LIN {X 0,Y 312.596,Z 485.644,A -85,B 0,C 180,E1 -15608.66,E2 -15608.66} C_VEL
LIN {X 0,Y 312.546,Z 485.552,A -85,B 0,C 180,E1 -15612.421,E2 -15612.421} C_VEL
LIN {X 0,Y 312.486,Z 485.523,A -85,B 0,C 180,E1 -15616.028,E2 -15616.028} C_VEL
LIN {X 0,Y 312.5,Z 485.561,A -85,B 0,C 180,E1 -15619.874,E2 -15619.874} C_VEL
LIN {X 0,Y 312.531,Z 485.556,A -85,B 0,C 180,E1 -15624.05,E2 -15624.05} C_VEL
LIN {X 0,Y 312.499,Z 485.544,A -85,B 0,C 180,E1 -15627.333,E2 -15627.333} C_VEL
LIN {X 0,Y 312.547,Z 485.546,A -85,B 0,C 180,E1 -15631.275,E2 -15631.275} C_VEL
LIN {X 0,Y 312.58,Z 485.536,A -85,B 0,C 180,E1 -15634.71,E2 -15634.71} C_VEL
LIN {X 0,Y 312.531,Z 485.541,A -85,B 0,C 180,E1 -15638.912,E2 -15638.912} C_VEL
LIN {X 0,Y 312.631,Z 485.51,A -85,B 0,C 180,E1 -15641.656,E2 -15641.656} C_VEL
LIN {X 0,Y 312.687,Z 485.534,A -85,B 0,C 180,E1 -15645.686,E2 -15645.686} C_VEL
LIN {X 0,Y 312.691,Z 485.521,A -85,B 0,C 180,E1 -15649.642,E2 -15649.642} C_VEL
LIN {X 0,Y 312.847,Z 485.516,A -85,B 0,C 180,E1 -15652.254,E2 -15652.254} C_VEL
LIN {X 0,Y 312.712,Z 485.516,A -85,B 0,C 180,E1 -15654.842,E2 -15654.842} C_VEL
LIN {X 0,Y 312.985,Z 485.5,A -85,B 0,C 180,E1 -15658.713,E2 -15658.713} C_VEL
LIN {X 0,Y 313.114,Z 485.481,A -85,B 0,C 180,E1 -15660,E2 -15660} C_VEL
LIN {X 0,Y 312.931,Z 485.487,A -85,B 0,C 180,E1 -15662.575,E2 -15662.575} C_VEL
LIN {X 0,Y 312.886,Z 485.51,A -85,B 0,C 180,E1 -15666.555,E2 -15666.555} C_VEL
LIN {X 0,Y 312.76,Z 485.507,A -85,B 0,C 180,E1 -15669.05,E2 -15669.05} C_VEL
LIN {X 0,Y 312.628,Z 485.542,A -85,B 0,C 180,E1 -15672.991,E2 -15672.991} C_VEL
LIN {X 0,Y 312.632,Z 485.527,A -85,B 0,C 180,E1 -15675.65,E2 -15675.65} C_VEL
LIN {X 0,Y 312.603,Z 485.546,A -85,B 0,C 180,E1 -15679.226,E2 -15679.226} C_VEL
LIN {X 0,Y 312.523,Z 485.543,A -85,B 0,C 180,E1 -15682.782,E2 -15682.782} C_VEL
LIN {X 0,Y 312.597,Z 485.545,A -85,B 0,C 180,E1 -15685.936,E2 -15685.936} C_VEL
LIN {X 0,Y 312.54,Z 485.51,A -85,B 0,C 180,E1 -15689.651,E2 -15689.651} C_VEL
LIN {X 0,Y 312.515,Z 485.544,A -85,B 0,C 180,E1 -15693.69,E2 -15693.69} C_VEL
LIN {X 0,Y 312.516,Z 485.547,A -85,B 0,C 180,E1 -15697.387,E2 -15697.387} C_VEL
LIN {X 0,Y 312.486,Z 485.524,A -85,B 0,C 180,E1 -15700.71,E2 -15700.71} C_VEL
LIN {X 0,Y 312.47,Z 485.562,A -85,B 0,C 180,E1 -15704.207,E2 -15704.207} C_VEL
LIN {X 0,Y 312.483,Z 485.536,A -85,B 0,C 180,E1 -15707.919,E2 -15707.919} C_VEL
LIN {X 0,Y 312.533,Z 485.543,A -85,B 0,C 180,E1 -15711.911,E2 -15711.911} C_VEL
LIN {X 0,Y 312.505,Z 485.487,A -85,B 0,C 180,E1 -15715.791,E2 -15715.791} C_VEL
LIN {X 0,Y 312.524,Z 485.55,A -85,B 0,C 180,E1 -15718.855,E2 -15718.855} C_VEL
LIN {X 0,Y 312.573,Z 485.515,A -85,B 0,C 180,E1 -15721.825,E2 -15721.825} C_VEL
LIN {X 0,Y 312.627,Z 485.658,A -85,B 0,C 180,E1 -15724.403,E2 -15724.403} C_VEL
LIN {X 0,Y 312.857,Z 486.708,A -85,B 0,C 180,E1 -15724.641,E2 -15724.641} C_VEL
LIN {X 0,Y 321.986,Z 506.318,A -85,B 0,C 180,E1 -15725.936,E2 -15725.936} C_VEL
LIN {X 0,Y 324.819,Z 512.869,A -85,B 0,C 180,E1 -15726.326,E2 -15726.326} C_VEL
LIN {X 0,Y 324.111,Z 565.204,A -85,B 0,C 180,E1 -15727.522,E2 -15727.522} C_VEL
LIN {X 0,Y 323.904,Z 578.235,A -85,B 0,C 180,E1 -15728.002,E2 -15728.002} C_VEL
LIN {X 0,Y 323.301,Z 591.093,A -85,B 0,C 180,E1 -15728.731,E2 -15728.731} C_VEL
LIN {X 0,Y 322.411,Z 603.924,A -85,B 0,C 180,E1 -15729.754,E2 -15729.754} C_VEL
LIN {X 0,Y 321.259,Z 614.593,A -85,B 0,C 180,E1 -15730.844,E2 -15730.844} C_VEL
LIN {X 0,Y 319.962,Z 625.427,A -85,B 0,C 180,E1 -15732.256,E2 -15732.256} C_VEL
LIN {X 0,Y 318.575,Z 635.942,A -85,B 0,C 180,E1 -15733.993,E2 -15733.993} C_VEL
LIN {X 0,Y 317.492,Z 643.676,A -85,B 0,C 180,E1 -15735.58,E2 -15735.58} C_VEL
LIN {X 0,Y 316.22,Z 651.351,A -85,B 0,C 180,E1 -15737.518,E2 -15737.518} C_VEL
LIN {X 0,Y 315.27,Z 657.101,A -85,B 0,C 180,E1 -15739.336,E2 -15739.336} C_VEL
LIN {X 0,Y 314.62,Z 661.367,A -85,B 0,C 180,E1 -15741.004,E2 -15741.004} C_VEL
LIN {X 0,Y 313.791,Z 665.259,A -85,B 0,C 180,E1 -15742.924,E2 -15742.924} C_VEL
LIN {X 0,Y 313.2,Z 668.127,A -85,B 0,C 180,E1 -15744.85,E2 -15744.85} C_VEL
LIN {X 0,Y 313.113,Z 669.472,A -85,B 0,C 180,E1 -15746.139,E2 -15746.139} C_VEL
LIN {X 0,Y 312.916,Z 671.03,A -85,B 0,C 180,E1 -15748.713,E2 -15748.713} C_VEL
LIN {X 0,Y 312.881,Z 671.257,A -85,B 0,C 180,E1 -15750,E2 -15750} C_VEL
LIN {X 0,Y 312.979,Z 670.503,A -85,B 0,C 180,E1 -15752.574,E2 -15752.574} C_VEL
LIN {X 0,Y 313.109,Z 669.563,A -85,B 0,C 180,E1 -15753.861,E2 -15753.861} C_VEL
LIN {X 0,Y 313.188,Z 668.259,A -85,B 0,C 180,E1 -15755.15,E2 -15755.15} C_VEL
LIN {X 0,Y 313.784,Z 665.44,A -85,B 0,C 180,E1 -15757.076,E2 -15757.076} C_VEL
LIN {X 0,Y 314.595,Z 661.613,A -85,B 0,C 180,E1 -15758.997,E2 -15758.997} C_VEL
LIN {X 0,Y 315.35,Z 656.533,A -85,B 0,C 180,E1 -15760.984,E2 -15760.984} C_VEL
LIN {X 0,Y 316.401,Z 650.502,A -85,B 0,C 180,E1 -15762.833,E2 -15762.833} C_VEL
LIN {X 0,Y 317.693,Z 642.72,A -85,B 0,C 180,E1 -15764.738,E2 -15764.738} C_VEL
LIN {X 0,Y 319.028,Z 633.047,A -85,B 0,C 180,E1 -15766.641,E2 -15766.641} C_VEL
LIN {X 0,Y 320.237,Z 624.003,A -85,B 0,C 180,E1 -15768.058,E2 -15768.058} C_VEL
LIN {X 0,Y 321.536,Z 613.493,A -85,B 0,C 180,E1 -15769.379,E2 -15769.379} C_VEL
LIN {X 0,Y 322.612,Z 601.973,A -85,B 0,C 180,E1 -15770.533,E2 -15770.533} C_VEL
LIN {X 0,Y 323.532,Z 590.691,A -85,B 0,C 180,E1 -15771.395,E2 -15771.395} C_VEL
LIN {X 0,Y 323.935,Z 578.331,A -85,B 0,C 180,E1 -15772.105,E2 -15772.105} C_VEL
LIN {X 0,Y 324.132,Z 566.47,A -85,B 0,C 180,E1 -15772.554,E2 -15772.554} C_VEL
LIN {X 0,Y 324.608,Z 528.424,A -85,B 0,C 180,E1 -15773.435,E2 -15773.435} C_VEL
LIN {X 0,Y 324.851,Z 512.955,A -85,B 0,C 180,E1 -15773.784,E2 -15773.784} C_VEL
LIN {X 0,Y 316.427,Z 494.129,A -85,B 0,C 180,E1 -15774.953,E2 -15774.953} C_VEL
LIN {X 0,Y 312.807,Z 486.547,A -85,B 0,C 180,E1 -15775.491,E2 -15775.491} C_VEL
LIN {X 0,Y 312.593,Z 485.593,A -85,B 0,C 180,E1 -15775.765,E2 -15775.765} C_VEL
LIN {X 0,Y 312.538,Z 485.545,A -85,B 0,C 180,E1 -15779.65,E2 -15779.65} C_VEL
LIN {X 0,Y 312.519,Z 485.552,A -85,B 0,C 180,E1 -15783.688,E2 -15783.688} C_VEL
LIN {X 0,Y 312.524,Z 485.539,A -85,B 0,C 180,E1 -15787.384,E2 -15787.384} C_VEL
LIN {X 0,Y 312.488,Z 485.554,A -85,B 0,C 180,E1 -15790.708,E2 -15790.708} C_VEL
LIN {X 0,Y 312.47,Z 485.55,A -85,B 0,C 180,E1 -15794.205,E2 -15794.205} C_VEL
LIN {X 0,Y 312.482,Z 485.55,A -85,B 0,C 180,E1 -15797.917,E2 -15797.917} C_VEL
LIN {X 0,Y 312.473,Z 485.529,A -85,B 0,C 180,E1 -15799.056,E2 -15799.056} C_VEL
LIN {X 0,Y 311.84,Z 485.603,A -85,B 0,C 180,E1 -15800.131,E2 -15800.131} C_VEL
LIN {X 0,Y 308.981,Z 485.976,A -85,B 0,C 180,E1 -15801.881,E2 -15801.881} C_VEL
LIN {X 0,Y 306.549,Z 486.296,A -85,B 0,C 180,E1 -15803.299,E2 -15803.299} C_VEL
LIN {X 0,Y 305.525,Z 486.427,A -85,B 0,C 180,E1 -15804.398,E2 -15804.398} C_VEL
LIN {X 0,Y 305.454,Z 486.437,A -85,B 0,C 180,E1 -15804.771,E2 -15804.771} C_VEL
LIN {X 0,Y 305.446,Z 486.391,A -85,B 0,C 180,E1 -15808.354,E2 -15808.354} C_VEL
LIN {X 0,Y 305.515,Z 486.394,A -85,B 0,C 180,E1 -15811.113,E2 -15811.113} C_VEL
LIN {X 0,Y 305.566,Z 486.421,A -85,B 0,C 180,E1 -15814.087,E2 -15814.087} C_VEL
LIN {X 0,Y 305.477,Z 486.422,A -85,B 0,C 180,E1 -15818.401,E2 -15818.401} C_VEL
LIN {X 0,Y 305.573,Z 486.422,A -85,B 0,C 180,E1 -15821.216,E2 -15821.216} C_VEL
LIN {X 0,Y 305.642,Z 486.404,A -85,B 0,C 180,E1 -15825.349,E2 -15825.349} C_VEL
LIN {X 0,Y 305.631,Z 486.4,A -85,B 0,C 180,E1 -15829.399,E2 -15829.399} C_VEL
LIN {X 0,Y 305.807,Z 486.385,A -85,B 0,C 180,E1 -15832.074,E2 -15832.074} C_VEL
LIN {X 0,Y 305.683,Z 486.404,A -85,B 0,C 180,E1 -15834.723,E2 -15834.723} C_VEL
LIN {X 0,Y 305.952,Z 486.36,A -85,B 0,C 180,E1 -15838.684,E2 -15838.684} C_VEL
LIN {X 0,Y 305.952,Z 486.372,A -85,B 0,C 180,E1 -15841.316,E2 -15841.316} C_VEL
LIN {X 0,Y 305.838,Z 486.384,A -85,B 0,C 180,E1 -15846.598,E2 -15846.598} C_VEL
LIN {X 0,Y 305.697,Z 486.399,A -85,B 0,C 180,E1 -15849.261,E2 -15849.261} C_VEL
LIN {X 0,Y 305.582,Z 486.417,A -85,B 0,C 180,E1 -15853.296,E2 -15853.296} C_VEL
LIN {X 0,Y 305.587,Z 486.411,A -85,B 0,C 180,E1 -15856.02,E2 -15856.02} C_VEL
LIN {X 0,Y 305.553,Z 486.39,A -85,B 0,C 180,E1 -15859.436,E2 -15859.436} C_VEL
LIN {X 0,Y 305.48,Z 486.433,A -85,B 0,C 180,E1 -15863.04,E2 -15863.04} C_VEL
LIN {X 0,Y 305.542,Z 486.401,A -85,B 0,C 180,E1 -15866.227,E2 -15866.227} C_VEL
LIN {X 0,Y 305.491,Z 486.426,A -85,B 0,C 180,E1 -15869.051,E2 -15869.051} C_VEL
LIN {X 0,Y 305.439,Z 486.427,A -85,B 0,C 180,E1 -15871.953,E2 -15871.953} C_VEL
LIN {X 0,Y 305.458,Z 486.433,A -85,B 0,C 180,E1 -15875.114,E2 -15875.114} C_VEL
LIN {X 0,Y 305.436,Z 486.427,A -85,B 0,C 180,E1 -15878.527,E2 -15878.527} C_VEL
LIN {X 0,Y 305.458,Z 486.409,A -85,B 0,C 180,E1 -15882.588,E2 -15882.588} C_VEL
LIN {X 0,Y 305.488,Z 486.426,A -85,B 0,C 180,E1 -15886.357,E2 -15886.357} C_VEL
LIN {X 0,Y 305.483,Z 486.408,A -85,B 0,C 180,E1 -15889.897,E2 -15889.897} C_VEL
LIN {X 0,Y 305.571,Z 486.704,A -85,B 0,C 180,E1 -15890.807,E2 -15890.807} C_VEL
LIN {X 0,Y 309.057,Z 500.296,A -85,B 0,C 180,E1 -15894.465,E2 -15894.465} C_VEL
LIN {X 0,Y 312.291,Z 514.772,A -85,B 0,C 180,E1 -15898.065,E2 -15898.065} C_VEL
LIN {X 0,Y 312.888,Z 518.28,A -85,B 0,C 180,E1 -15898.895,E2 -15898.895} C_VEL
LIN {X 0,Y 310.582,Z 534.816,A -85,B 0,C 180,E1 -15902.4,E2 -15902.4} C_VEL
LIN {X 0,Y 309.847,Z 540.998,A -85,B 0,C 180,E1 -15903.672,E2 -15903.672} C_VEL
LIN {X 0,Y 313.493,Z 569.986,A -85,B 0,C 180,E1 -15904.736,E2 -15904.736} C_VEL
LIN {X 0,Y 316.513,Z 601.665,A -85,B 0,C 180,E1 -15905.751,E2 -15905.751} C_VEL
LIN {X 0,Y 316.362,Z 614.838,A -85,B 0,C 180,E1 -15906.058,E2 -15906.058} C_VEL
LIN {X 0,Y 315.444,Z 652.112,A -85,B 0,C 180,E1 -15906.923,E2 -15906.923} C_VEL
LIN {X 0,Y 314.652,Z 665.36,A -85,B 0,C 180,E1 -15907.469,E2 -15907.469} C_VEL
LIN {X 0,Y 313.462,Z 677.536,A -85,B 0,C 180,E1 -15908.202,E2 -15908.202} C_VEL
LIN {X 0,Y 311.89,Z 689.848,A -85,B 0,C 180,E1 -15909.213,E2 -15909.213} C_VEL
LIN {X 0,Y 310.154,Z 701.52,A -85,B 0,C 180,E1 -15910.475,E2 -15910.475} C_VEL
LIN {X 0,Y 308.633,Z 712.087,A -85,B 0,C 180,E1 -15911.926,E2 -15911.926} C_VEL
LIN {X 0,Y 307.351,Z 720.759,A -85,B 0,C 180,E1 -15913.392,E2 -15913.392} C_VEL
LIN {X 0,Y 306.018,Z 729.046,A -85,B 0,C 180,E1 -15915.091,E2 -15915.091} C_VEL
LIN {X 0,Y 305.136,Z 736.674,A -85,B 0,C 180,E1 -15917.023,E2 -15917.023} C_VEL
LIN {X 0,Y 304.49,Z 744.006,A -85,B 0,C 180,E1 -15919.36,E2 -15919.36} C_VEL
LIN {X 0,Y 304.349,Z 748.934,A -85,B 0,C 180,E1 -15921.368,E2 -15921.368} C_VEL
LIN {X 0,Y 304.476,Z 752.737,A -85,B 0,C 180,E1 -15923.373,E2 -15923.373} C_VEL
LIN {X 0,Y 304.614,Z 754.709,A -85,B 0,C 180,E1 -15924.705,E2 -15924.705} C_VEL
LIN {X 0,Y 304.878,Z 756.212,A -85,B 0,C 180,E1 -15926.035,E2 -15926.035} C_VEL
LIN {X 0,Y 305.27,Z 757.949,A -85,B 0,C 180,E1 -15928.681,E2 -15928.681} C_VEL
LIN {X 0,Y 305.514,Z 758.207,A -85,B 0,C 180,E1 -15930,E2 -15930} C_VEL
LIN {X 0,Y 305.272,Z 757.943,A -85,B 0,C 180,E1 -15931.319,E2 -15931.319} C_VEL
LIN {X 0,Y 304.881,Z 756.2,A -85,B 0,C 180,E1 -15933.965,E2 -15933.965} C_VEL
LIN {X 0,Y 304.621,Z 754.691,A -85,B 0,C 180,E1 -15935.295,E2 -15935.295} C_VEL
LIN {X 0,Y 304.457,Z 752.124,A -85,B 0,C 180,E1 -15936.973,E2 -15936.973} C_VEL
LIN {X 0,Y 304.367,Z 747.393,A -85,B 0,C 180,E1 -15939.301,E2 -15939.301} C_VEL
LIN {X 0,Y 304.714,Z 741.027,A -85,B 0,C 180,E1 -15941.643,E2 -15941.643} C_VEL
LIN {X 0,Y 305.401,Z 734.135,A -85,B 0,C 180,E1 -15943.643,E2 -15943.643} C_VEL
LIN {X 0,Y 306.5,Z 725.676,A -85,B 0,C 180,E1 -15945.622,E2 -15945.622} C_VEL
LIN {X 0,Y 307.797,Z 716.984,A -85,B 0,C 180,E1 -15947.267,E2 -15947.267} C_VEL
LIN {X 0,Y 309.411,Z 706.336,A -85,B 0,C 180,E1 -15948.885,E2 -15948.885} C_VEL
LIN {X 0,Y 311.225,Z 694.405,A -85,B 0,C 180,E1 -15950.315,E2 -15950.315} C_VEL
LIN {X 0,Y 312.822,Z 682.418,A -85,B 0,C 180,E1 -15951.412,E2 -15951.412} C_VEL
LIN {X 0,Y 314.215,Z 669.976,A -85,B 0,C 180,E1 -15952.261,E2 -15952.261} C_VEL
LIN {X 0,Y 315.133,Z 657.164,A -85,B 0,C 180,E1 -15952.885,E2 -15952.885} C_VEL
LIN {X 0,Y 315.641,Z 643.669,A -85,B 0,C 180,E1 -15953.279,E2 -15953.279} C_VEL
LIN {X 0,Y 316.552,Z 602.566,A -85,B 0,C 180,E1 -15954.202,E2 -15954.202} C_VEL
LIN {X 0,Y 313.303,Z 568.848,A -85,B 0,C 180,E1 -15955.284,E2 -15955.284} C_VEL
LIN {X 0,Y 309.777,Z 541.191,A -85,B 0,C 180,E1 -15956.291,E2 -15956.291} C_VEL
LIN {X 0,Y 310.569,Z 534.66,A -85,B 0,C 180,E1 -15957.612,E2 -15957.612} C_VEL
LIN {X 0,Y 312.701,Z 519.8,A -85,B 0,C 180,E1 -15960.75,E2 -15960.75} C_VEL
LIN {X 0,Y 312.718,Z 517.094,A -85,B 0,C 180,E1 -15961.349,E2 -15961.349} C_VEL
LIN {X 0,Y 310.298,Z 505.665,A -85,B 0,C 180,E1 -15964.147,E2 -15964.147} C_VEL
LIN {X 0,Y 307.275,Z 493.295,A -85,B 0,C 180,E1 -15967.344,E2 -15967.344} C_VEL
LIN {X 0,Y 305.526,Z 486.498,A -85,B 0,C 180,E1 -15969.271,E2 -15969.271} C_VEL
LIN {X 0,Y 305.505,Z 486.432,A -85,B 0,C 180,E1 -15972.596,E2 -15972.596} C_VEL
LIN {X 0,Y 305.446,Z 486.399,A -85,B 0,C 180,E1 -15976.348,E2 -15976.348} C_VEL
LIN {X 0,Y 305.454,Z 486.438,A -85,B 0,C 180,E1 -15979.892,E2 -15979.892} C_VEL
LIN {X 0,Y 305.476,Z 486.432,A -85,B 0,C 180,E1 -15983.631,E2 -15983.631} C_VEL
LIN {X 0,Y 305.46,Z 486.418,A -85,B 0,C 180,E1 -15986.483,E2 -15986.483} C_VEL
LIN {X 0,Y 305.458,Z 486.436,A -85,B 0,C 180,E1 -15989.59,E2 -15989.59} C_VEL
LIN {X 0,Y 305.516,Z 486.404,A -85,B 0,C 180,E1 -15992.608,E2 -15992.608} C_VEL
LIN {X 0,Y 305.5,Z 486.426,A -85,B 0,C 180,E1 -15995.538,E2 -15995.538} C_VEL
LIN {X 0,Y 305.5,Z 486.404,A -85,B 0,C 180,E1 -15999.814,E2 -15999.814} C_VEL
LIN {X 0,Y 305.567,Z 486.398,A -85,B 0,C 180,E1 -16002.603,E2 -16002.603} C_VEL
LIN {X 0,Y 305.642,Z 486.411,A -85,B 0,C 180,E1 -16005.349,E2 -16005.349} C_VEL
LIN {X 0,Y 305.628,Z 486.399,A -85,B 0,C 180,E1 -16009.399,E2 -16009.399} C_VEL
LIN {X 0,Y 305.791,Z 486.394,A -85,B 0,C 180,E1 -16012.074,E2 -16012.074} C_VEL
LIN {X 0,Y 305.683,Z 486.392,A -85,B 0,C 180,E1 -16014.723,E2 -16014.723} C_VEL
LIN {X 0,Y 305.952,Z 486.376,A -85,B 0,C 180,E1 -16018.684,E2 -16018.684} C_VEL
LIN {X 0,Y 305.952,Z 486.363,A -85,B 0,C 180,E1 -16021.316,E2 -16021.316} C_VEL
LIN {X 0,Y 305.684,Z 486.405,A -85,B 0,C 180,E1 -16025.277,E2 -16025.277} C_VEL
LIN {X 0,Y 305.791,Z 486.388,A -85,B 0,C 180,E1 -16027.926,E2 -16027.926} C_VEL
LIN {X 0,Y 305.596,Z 486.414,A -85,B 0,C 180,E1 -16031.945,E2 -16031.945} C_VEL
LIN {X 0,Y 305.631,Z 486.401,A -85,B 0,C 180,E1 -16035.035,E2 -16035.035} C_VEL
LIN {X 0,Y 305.573,Z 486.422,A -85,B 0,C 180,E1 -16038.784,E2 -16038.784} C_VEL
LIN {X 0,Y 305.48,Z 486.421,A -85,B 0,C 180,E1 -16043.04,E2 -16043.04} C_VEL
LIN {X 0,Y 305.542,Z 486.424,A -85,B 0,C 180,E1 -16046.228,E2 -16046.228} C_VEL
LIN {X 0,Y 305.49,Z 486.396,A -85,B 0,C 180,E1 -16049.05,E2 -16049.05} C_VEL
LIN {X 0,Y 305.438,Z 486.395,A -85,B 0,C 180,E1 -16051.953,E2 -16051.953} C_VEL
LIN {X 0,Y 305.458,Z 486.436,A -85,B 0,C 180,E1 -16055.114,E2 -16055.114} C_VEL
LIN {X 0,Y 305.436,Z 486.411,A -85,B 0,C 180,E1 -16058.527,E2 -16058.527} C_VEL
LIN {X 0,Y 305.456,Z 486.427,A -85,B 0,C 180,E1 -16062.587,E2 -16062.587} C_VEL
LIN {X 0,Y 305.44,Z 486.417,A -85,B 0,C 180,E1 -16066.349,E2 -16066.349} C_VEL
LIN {X 0,Y 305.456,Z 486.436,A -85,B 0,C 180,E1 -16069.893,E2 -16069.893} C_VEL
LIN {X 0,Y 305.48,Z 486.379,A -85,B 0,C 180,E1 -16073.632,E2 -16073.632} C_VEL
LIN {X 0,Y 305.464,Z 486.368,A -85,B 0,C 180,E1 -16076.484,E2 -16076.484} C_VEL
LIN {X 0,Y 305.464,Z 486.44,A -85,B 0,C 180,E1 -16079.592,E2 -16079.592} C_VEL
LIN {X 0,Y 305.521,Z 486.385,A -85,B 0,C 180,E1 -16083.262,E2 -16083.262} C_VEL
LIN {X 0,Y 305.606,Z 486.712,A -85,B 0,C 180,E1 -16083.841,E2 -16083.841} C_VEL
LIN {X 0,Y 305.872,Z 487.768,A -85,B 0,C 180,E1 -16084.024,E2 -16084.024} C_VEL
LIN {X 0,Y 314.752,Z 506.474,A -85,B 0,C 180,E1 -16085.322,E2 -16085.322} C_VEL
LIN {X 0,Y 318.442,Z 514.916,A -85,B 0,C 180,E1 -16085.847,E2 -16085.847} C_VEL
LIN {X 0,Y 317.657,Z 559.958,A -85,B 0,C 180,E1 -16086.878,E2 -16086.878} C_VEL
LIN {X 0,Y 317.511,Z 574.854,A -85,B 0,C 180,E1 -16087.33,E2 -16087.33} C_VEL
LIN {X 0,Y 317.049,Z 587.08,A -85,B 0,C 180,E1 -16087.948,E2 -16087.948} C_VEL
LIN {X 0,Y 316.25,Z 599.866,A -85,B 0,C 180,E1 -16088.866,E2 -16088.866} C_VEL
LIN {X 0,Y 315.259,Z 611.317,A -85,B 0,C 180,E1 -16089.955,E2 -16089.955} C_VEL
LIN {X 0,Y 314.025,Z 620.729,A -85,B 0,C 180,E1 -16091.064,E2 -16091.064} C_VEL
LIN {X 0,Y 312.889,Z 629.558,A -85,B 0,C 180,E1 -16092.349,E2 -16092.349} C_VEL
LIN {X 0,Y 311.603,Z 638.599,A -85,B 0,C 180,E1 -16093.961,E2 -16093.961} C_VEL
LIN {X 0,Y 310.23,Z 647.36,A -85,B 0,C 180,E1 -16095.905,E2 -16095.905} C_VEL
LIN {X 0,Y 309.156,Z 653.537,A -85,B 0,C 180,E1 -16097.595,E2 -16097.595} C_VEL
LIN {X 0,Y 308.208,Z 659.146,A -85,B 0,C 180,E1 -16099.489,E2 -16099.489} C_VEL
LIN {X 0,Y 307.32,Z 663.758,A -85,B 0,C 180,E1 -16101.452,E2 -16101.452} C_VEL
LIN {X 0,Y 306.565,Z 667.293,A -85,B 0,C 180,E1 -16103.418,E2 -16103.418} C_VEL
LIN {X 0,Y 306.198,Z 669.116,A -85,B 0,C 180,E1 -16104.732,E2 -16104.732} C_VEL
LIN {X 0,Y 306.101,Z 670.461,A -85,B 0,C 180,E1 -16106.05,E2 -16106.05} C_VEL
LIN {X 0,Y 305.893,Z 672.018,A -85,B 0,C 180,E1 -16108.684,E2 -16108.684} C_VEL
LIN {X 0,Y 305.854,Z 672.245,A -85,B 0,C 180,E1 -16110,E2 -16110} C_VEL
LIN {X 0,Y 305.972,Z 671.489,A -85,B 0,C 180,E1 -16112.633,E2 -16112.633} C_VEL
LIN {X 0,Y 306.096,Z 670.551,A -85,B 0,C 180,E1 -16113.95,E2 -16113.95} C_VEL
LIN {X 0,Y 306.186,Z 669.247,A -85,B 0,C 180,E1 -16115.268,E2 -16115.268} C_VEL
LIN {X 0,Y 306.811,Z 666.428,A -85,B 0,C 180,E1 -16117.238,E2 -16117.238} C_VEL
LIN {X 0,Y 307.655,Z 662.6,A -85,B 0,C 180,E1 -16119.201,E2 -16119.201} C_VEL
LIN {X 0,Y 308.453,Z 657.52,A -85,B 0,C 180,E1 -16121.233,E2 -16121.233} C_VEL
LIN {X 0,Y 309.552,Z 651.488,A -85,B 0,C 180,E1 -16123.122,E2 -16123.122} C_VEL
LIN {X 0,Y 310.901,Z 643.706,A -85,B 0,C 180,E1 -16125.067,E2 -16125.067} C_VEL
LIN {X 0,Y 312.299,Z 634.032,A -85,B 0,C 180,E1 -16127.01,E2 -16127.01} C_VEL
LIN {X 0,Y 313.561,Z 624.987,A -85,B 0,C 180,E1 -16128.456,E2 -16128.456} C_VEL
LIN {X 0,Y 314.915,Z 614.476,A -85,B 0,C 180,E1 -16129.804,E2 -16129.804} C_VEL
LIN {X 0,Y 316.04,Z 602.955,A -85,B 0,C 180,E1 -16130.98,E2 -16130.98} C_VEL
LIN {X 0,Y 317.003,Z 591.671,A -85,B 0,C 180,E1 -16131.858,E2 -16131.858} C_VEL
LIN {X 0,Y 317.414,Z 579.503,A -85,B 0,C 180,E1 -16132.575,E2 -16132.575} C_VEL
LIN {X 0,Y 317.65,Z 566.728,A -85,B 0,C 180,E1 -16133.061,E2 -16133.061} C_VEL
LIN {X 0,Y 318.156,Z 528.434,A -85,B 0,C 180,E1 -16133.963,E2 -16133.963} C_VEL
LIN {X 0,Y 318.389,Z 514.776,A -85,B 0,C 180,E1 -16134.276,E2 -16134.276} C_VEL
LIN {X 0,Y 309.566,Z 495.231,A -85,B 0,C 180,E1 -16135.544,E2 -16135.544} C_VEL
LIN {X 0,Y 305.71,Z 487.248,A -85,B 0,C 180,E1 -16136.153,E2 -16136.153} C_VEL
LIN {X 0,Y 305.539,Z 486.47,A -85,B 0,C 180,E1 -16136.411,E2 -16136.411} C_VEL
LIN {X 0,Y 305.487,Z 486.407,A -85,B 0,C 180,E1 -16139.046,E2 -16139.046} C_VEL
LIN {X 0,Y 305.441,Z 486.425,A -85,B 0,C 180,E1 -16141.952,E2 -16141.952} C_VEL
LIN {X 0,Y 305.461,Z 486.433,A -85,B 0,C 180,E1 -16145.112,E2 -16145.112} C_VEL
LIN {X 0,Y 305.448,Z 486.432,A -85,B 0,C 180,E1 -16148.528,E2 -16148.528} C_VEL
LIN {X 0,Y 305.456,Z 486.41,A -85,B 0,C 180,E1 -16152.586,E2 -16152.586} C_VEL
LIN {X 0,Y 305.44,Z 486.439,A -85,B 0,C 180,E1 -16156.347,E2 -16156.347} C_VEL
LIN {X 0,Y 305.454,Z 486.396,A -85,B 0,C 180,E1 -16159.891,E2 -16159.891} C_VEL
LIN {X 0,Y 305.476,Z 486.434,A -85,B 0,C 180,E1 -16163.631,E2 -16163.631} C_VEL
LIN {X 0,Y 305.454,Z 486.437,A -85,B 0,C 180,E1 -16164.771,E2 -16164.771} C_VEL
LIN {X 0,Y 304.824,Z 486.515,A -85,B 0,C 180,E1 -16165.871,E2 -16165.871} C_VEL
LIN {X 0,Y 302,Z 486.845,A -85,B 0,C 180,E1 -16167.664,E2 -16167.664} C_VEL
LIN {X 0,Y 299.575,Z 487.128,A -85,B 0,C 180,E1 -16169.117,E2 -16169.117} C_VEL
LIN {X 0,Y 298.519,Z 487.255,A -85,B 0,C 180,E1 -16170.243,E2 -16170.243} C_VEL
LIN {X 0,Y 298.426,Z 487.268,A -85,B 0,C 180,E1 -16170.625,E2 -16170.625} C_VEL
LIN {X 0,Y 298.479,Z 487.301,A -85,B 0,C 180,E1 -16173.474,E2 -16173.474} C_VEL
LIN {X 0,Y 298.426,Z 487.302,A -85,B 0,C 180,E1 -16176.699,E2 -16176.699} C_VEL
LIN {X 0,Y 298.519,Z 487.299,A -85,B 0,C 180,E1 -16180.755,E2 -16180.755} C_VEL
LIN {X 0,Y 298.587,Z 487.279,A -85,B 0,C 180,E1 -16184.994,E2 -16184.994} C_VEL
LIN {X 0,Y 298.587,Z 487.28,A -85,B 0,C 180,E1 -16189.146,E2 -16189.146} C_VEL
LIN {X 0,Y 298.753,Z 487.26,A -85,B 0,C 180,E1 -16191.886,E2 -16191.886} C_VEL
LIN {X 0,Y 298.654,Z 487.279,A -85,B 0,C 180,E1 -16194.599,E2 -16194.599} C_VEL
LIN {X 0,Y 298.918,Z 487.236,A -85,B 0,C 180,E1 -16198.653,E2 -16198.653} C_VEL
LIN {X 0,Y 298.918,Z 487.248,A -85,B 0,C 180,E1 -16201.347,E2 -16201.347} C_VEL
LIN {X 0,Y 298.782,Z 487.263,A -85,B 0,C 180,E1 -16206.754,E2 -16206.754} C_VEL
LIN {X 0,Y 298.628,Z 487.276,A -85,B 0,C 180,E1 -16209.482,E2 -16209.482} C_VEL
LIN {X 0,Y 298.545,Z 487.297,A -85,B 0,C 180,E1 -16213.616,E2 -16213.616} C_VEL
LIN {X 0,Y 298.542,Z 487.287,A -85,B 0,C 180,E1 -16216.409,E2 -16216.409} C_VEL
LIN {X 0,Y 298.491,Z 487.27,A -85,B 0,C 180,E1 -16219.647,E2 -16219.647} C_VEL
LIN {X 0,Y 298.45,Z 487.31,A -85,B 0,C 180,E1 -16223.598,E2 -16223.598} C_VEL
LIN {X 0,Y 298.484,Z 487.278,A -85,B 0,C 180,E1 -16226.575,E2 -16226.575} C_VEL
LIN {X 0,Y 298.416,Z 487.312,A -85,B 0,C 180,E1 -16229.642,E2 -16229.642} C_VEL
LIN {X 0,Y 298.391,Z 487.298,A -85,B 0,C 180,E1 -16232.801,E2 -16232.801} C_VEL
LIN {X 0,Y 298.44,Z 487.308,A -85,B 0,C 180,E1 -16236.808,E2 -16236.808} C_VEL
LIN {X 0,Y 298.385,Z 487.315,A -85,B 0,C 180,E1 -16241.089,E2 -16241.089} C_VEL
LIN {X 0,Y 298.414,Z 487.28,A -85,B 0,C 180,E1 -16245.048,E2 -16245.048} C_VEL
LIN {X 0,Y 298.449,Z 487.287,A -85,B 0,C 180,E1 -16248.751,E2 -16248.751} C_VEL
LIN {X 0,Y 298.484,Z 487.536,A -85,B 0,C 180,E1 -16250.183,E2 -16250.183} C_VEL
LIN {X 0,Y 301.581,Z 499.423,A -85,B 0,C 180,E1 -16253.512,E2 -16253.512} C_VEL
LIN {X 0,Y 304.298,Z 511.296,A -85,B 0,C 180,E1 -16256.595,E2 -16256.595} C_VEL
LIN {X 0,Y 305.956,Z 519.029,A -85,B 0,C 180,E1 -16258.524,E2 -16258.524} C_VEL
LIN {X 0,Y 305.188,Z 525.503,A -85,B 0,C 180,E1 -16259.943,E2 -16259.943} C_VEL
LIN {X 0,Y 303.156,Z 539.847,A -85,B 0,C 180,E1 -16263.032,E2 -16263.032} C_VEL
LIN {X 0,Y 306.583,Z 567.131,A -85,B 0,C 180,E1 -16264.079,E2 -16264.079} C_VEL
LIN {X 0,Y 309.547,Z 596.354,A -85,B 0,C 180,E1 -16265.063,E2 -16265.063} C_VEL
LIN {X 0,Y 310.121,Z 605.86,A -85,B 0,C 180,E1 -16265.346,E2 -16265.346} C_VEL
LIN {X 0,Y 308.915,Z 651.126,A -85,B 0,C 180,E1 -16266.406,E2 -16266.406} C_VEL
LIN {X 0,Y 308.097,Z 664.369,A -85,B 0,C 180,E1 -16266.962,E2 -16266.962} C_VEL
LIN {X 0,Y 306.858,Z 676.541,A -85,B 0,C 180,E1 -16267.708,E2 -16267.708} C_VEL
LIN {X 0,Y 305.245,Z 688.851,A -85,B 0,C 180,E1 -16268.739,E2 -16268.739} C_VEL
LIN {X 0,Y 303.453,Z 700.523,A -85,B 0,C 180,E1 -16270.025,E2 -16270.025} C_VEL
LIN {X 0,Y 302.03,Z 710.002,A -85,B 0,C 180,E1 -16271.34,E2 -16271.34} C_VEL
LIN {X 0,Y 300.471,Z 719.751,A -85,B 0,C 180,E1 -16273,E2 -16273} C_VEL
LIN {X 0,Y 299.049,Z 727.657,A -85,B 0,C 180,E1 -16274.648,E2 -16274.648} C_VEL
LIN {X 0,Y 298.464,Z 733.205,A -85,B 0,C 180,E1 -16276.034,E2 -16276.034} C_VEL
LIN {X 0,Y 297.706,Z 740.081,A -85,B 0,C 180,E1 -16278.079,E2 -16278.079} C_VEL
LIN {X 0,Y 297.286,Z 746.427,A -85,B 0,C 180,E1 -16280.475,E2 -16280.475} C_VEL
LIN {X 0,Y 297.355,Z 751.478,A -85,B 0,C 180,E1 -16283.06,E2 -16283.06} C_VEL
LIN {X 0,Y 297.529,Z 753.709,A -85,B 0,C 180,E1 -16284.578,E2 -16284.578} C_VEL
LIN {X 0,Y 297.804,Z 755.215,A -85,B 0,C 180,E1 -16285.94,E2 -16285.94} C_VEL
LIN {X 0,Y 298.213,Z 756.956,A -85,B 0,C 180,E1 -16288.65,E2 -16288.65} C_VEL
LIN {X 0,Y 298.482,Z 757.218,A -85,B 0,C 180,E1 -16290,E2 -16290} C_VEL
LIN {X 0,Y 298.214,Z 756.95,A -85,B 0,C 180,E1 -16291.35,E2 -16291.35} C_VEL
LIN {X 0,Y 297.808,Z 755.202,A -85,B 0,C 180,E1 -16294.06,E2 -16294.06} C_VEL
LIN {X 0,Y 297.538,Z 753.69,A -85,B 0,C 180,E1 -16295.421,E2 -16295.421} C_VEL
LIN {X 0,Y 297.344,Z 750.573,A -85,B 0,C 180,E1 -16297.469,E2 -16297.469} C_VEL
LIN {X 0,Y 297.286,Z 746.383,A -85,B 0,C 180,E1 -16299.525,E2 -16299.525} C_VEL
LIN {X 0,Y 297.716,Z 740.021,A -85,B 0,C 180,E1 -16301.92,E2 -16301.92} C_VEL
LIN {X 0,Y 298.465,Z 733.129,A -85,B 0,C 180,E1 -16303.966,E2 -16303.966} C_VEL
LIN {X 0,Y 299.523,Z 725.347,A -85,B 0,C 180,E1 -16305.841,E2 -16305.841} C_VEL
LIN {X 0,Y 300.949,Z 715.972,A -85,B 0,C 180,E1 -16307.673,E2 -16307.673} C_VEL
LIN {X 0,Y 302.701,Z 705.334,A -85,B 0,C 180,E1 -16309.32,E2 -16309.32} C_VEL
LIN {X 0,Y 304.553,Z 693.399,A -85,B 0,C 180,E1 -16310.781,E2 -16310.781} C_VEL
LIN {X 0,Y 306.223,Z 681.414,A -85,B 0,C 180,E1 -16311.897,E2 -16311.897} C_VEL
LIN {X 0,Y 307.643,Z 668.968,A -85,B 0,C 180,E1 -16312.763,E2 -16312.763} C_VEL
LIN {X 0,Y 308.595,Z 656.153,A -85,B 0,C 180,E1 -16313.398,E2 -16313.398} C_VEL
LIN {X 0,Y 309.118,Z 642.647,A -85,B 0,C 180,E1 -16313.8,E2 -16313.8} C_VEL
LIN {X 0,Y 309.969,Z 602.608,A -85,B 0,C 180,E1 -16314.723,E2 -16314.723} C_VEL
LIN {X 0,Y 306.904,Z 570.169,A -85,B 0,C 180,E1 -16315.791,E2 -16315.791} C_VEL
LIN {X 0,Y 303.113,Z 540.033,A -85,B 0,C 180,E1 -16316.925,E2 -16316.925} C_VEL
LIN {X 0,Y 305.667,Z 522.115,A -85,B 0,C 180,E1 -16320.767,E2 -16320.767} C_VEL
LIN {X 0,Y 305.918,Z 518.996,A -85,B 0,C 180,E1 -16321.457,E2 -16321.457} C_VEL
LIN {X 0,Y 303.682,Z 508.277,A -85,B 0,C 180,E1 -16324.139,E2 -16324.139} C_VEL
LIN {X 0,Y 301.137,Z 497.669,A -85,B 0,C 180,E1 -16326.933,E2 -16326.933} C_VEL
LIN {X 0,Y 298.468,Z 487.405,A -85,B 0,C 180,E1 -16329.852,E2 -16329.852} C_VEL
LIN {X 0,Y 298.457,Z 487.311,A -85,B 0,C 180,E1 -16333.115,E2 -16333.115} C_VEL
LIN {X 0,Y 298.399,Z 487.28,A -85,B 0,C 180,E1 -16336.92,E2 -16336.92} C_VEL
LIN {X 0,Y 298.395,Z 487.305,A -85,B 0,C 180,E1 -16341.007,E2 -16341.007} C_VEL
LIN {X 0,Y 298.414,Z 487.314,A -85,B 0,C 180,E1 -16343.929,E2 -16343.929} C_VEL
LIN {X 0,Y 298.39,Z 487.305,A -85,B 0,C 180,E1 -16347.983,E2 -16347.983} C_VEL
LIN {X 0,Y 298.458,Z 487.289,A -85,B 0,C 180,E1 -16351.904,E2 -16351.904} C_VEL
LIN {X 0,Y 298.479,Z 487.294,A -85,B 0,C 180,E1 -16354.923,E2 -16354.923} C_VEL
LIN {X 0,Y 298.431,Z 487.292,A -85,B 0,C 180,E1 -16359.314,E2 -16359.314} C_VEL
LIN {X 0,Y 298.527,Z 487.27,A -85,B 0,C 180,E1 -16362.179,E2 -16362.179} C_VEL
LIN {X 0,Y 298.587,Z 487.292,A -85,B 0,C 180,E1 -16364.994,E2 -16364.994} C_VEL
LIN {X 0,Y 298.584,Z 487.275,A -85,B 0,C 180,E1 -16369.146,E2 -16369.146} C_VEL
LIN {X 0,Y 298.735,Z 487.272,A -85,B 0,C 180,E1 -16371.885,E2 -16371.885} C_VEL
LIN {X 0,Y 298.653,Z 487.268,A -85,B 0,C 180,E1 -16374.599,E2 -16374.599} C_VEL
LIN {X 0,Y 298.918,Z 487.251,A -85,B 0,C 180,E1 -16378.653,E2 -16378.653} C_VEL
LIN {X 0,Y 298.918,Z 487.239,A -85,B 0,C 180,E1 -16381.347,E2 -16381.347} C_VEL
LIN {X 0,Y 298.783,Z 487.265,A -85,B 0,C 180,E1 -16386.754,E2 -16386.754} C_VEL
LIN {X 0,Y 298.629,Z 487.266,A -85,B 0,C 180,E1 -16389.482,E2 -16389.482} C_VEL
LIN {X 0,Y 298.545,Z 487.294,A -85,B 0,C 180,E1 -16393.616,E2 -16393.616} C_VEL
LIN {X 0,Y 298.542,Z 487.28,A -85,B 0,C 180,E1 -16396.409,E2 -16396.409} C_VEL
LIN {X 0,Y 298.492,Z 487.302,A -85,B 0,C 180,E1 -16399.648,E2 -16399.648} C_VEL
LIN {X 0,Y 298.424,Z 487.305,A -85,B 0,C 180,E1 -16403.601,E2 -16403.601} C_VEL
LIN {X 0,Y 298.485,Z 487.3,A -85,B 0,C 180,E1 -16406.575,E2 -16406.575} C_VEL
LIN {X 0,Y 298.416,Z 487.267,A -85,B 0,C 180,E1 -16409.642,E2 -16409.642} C_VEL
LIN {X 0,Y 298.391,Z 487.287,A -85,B 0,C 180,E1 -16412.801,E2 -16412.801} C_VEL
LIN {X 0,Y 298.44,Z 487.306,A -85,B 0,C 180,E1 -16416.808,E2 -16416.808} C_VEL
LIN {X 0,Y 298.384,Z 487.282,A -85,B 0,C 180,E1 -16421.088,E2 -16421.088} C_VEL
LIN {X 0,Y 298.386,Z 487.311,A -85,B 0,C 180,E1 -16425.042,E2 -16425.042} C_VEL
LIN {X 0,Y 298.385,Z 487.302,A -85,B 0,C 180,E1 -16428.913,E2 -16428.913} C_VEL
LIN {X 0,Y 298.423,Z 487.291,A -85,B 0,C 180,E1 -16432.244,E2 -16432.244} C_VEL
LIN {X 0,Y 298.407,Z 487.24,A -85,B 0,C 180,E1 -16435.582,E2 -16435.582} C_VEL
LIN {X 0,Y 298.396,Z 487.304,A -85,B 0,C 180,E1 -16438.792,E2 -16438.792} C_VEL
LIN {X 0,Y 298.485,Z 487.362,A -85,B 0,C 180,E1 -16443.001,E2 -16443.001} C_VEL
LIN {X 0,Y 298.682,Z 488.194,A -85,B 0,C 180,E1 -16443.305,E2 -16443.305} C_VEL
LIN {X 0,Y 307.424,Z 506.32,A -85,B 0,C 180,E1 -16444.659,E2 -16444.659} C_VEL
LIN {X 0,Y 311.906,Z 516.555,A -85,B 0,C 180,E1 -16445.323,E2 -16445.323} C_VEL
LIN {X 0,Y 311.162,Z 567.185,A -85,B 0,C 180,E1 -16446.531,E2 -16446.531} C_VEL
LIN {X 0,Y 310.871,Z 580.538,A -85,B 0,C 180,E1 -16447.043,E2 -16447.043} C_VEL
LIN {X 0,Y 310.239,Z 593.086,A -85,B 0,C 180,E1 -16447.789,E2 -16447.789} C_VEL
LIN {X 0,Y 309.263,Z 605.909,A -85,B 0,C 180,E1 -16448.852,E2 -16448.852} C_VEL
LIN {X 0,Y 308.017,Z 616.579,A -85,B 0,C 180,E1 -16449.986,E2 -16449.986} C_VEL
LIN {X 0,Y 306.602,Z 627.411,A -85,B 0,C 180,E1 -16451.456,E2 -16451.456} C_VEL
LIN {X 0,Y 305.087,Z 637.924,A -85,B 0,C 180,E1 -16453.265,E2 -16453.265} C_VEL
LIN {X 0,Y 303.899,Z 645.657,A -85,B 0,C 180,E1 -16454.92,E2 -16454.92} C_VEL
LIN {X 0,Y 302.512,Z 653.331,A -85,B 0,C 180,E1 -16456.943,E2 -16456.943} C_VEL
LIN {X 0,Y 301.467,Z 659.08,A -85,B 0,C 180,E1 -16458.842,E2 -16458.842} C_VEL
LIN {X 0,Y 300.745,Z 663.346,A -85,B 0,C 180,E1 -16460.585,E2 -16460.585} C_VEL
LIN {X 0,Y 299.847,Z 667.237,A -85,B 0,C 180,E1 -16462.593,E2 -16462.593} C_VEL
LIN {X 0,Y 299.198,Z 670.105,A -85,B 0,C 180,E1 -16464.609,E2 -16464.609} C_VEL
LIN {X 0,Y 299.089,Z 671.45,A -85,B 0,C 180,E1 -16465.958,E2 -16465.958} C_VEL
LIN {X 0,Y 298.87,Z 673.006,A -85,B 0,C 180,E1 -16468.653,E2 -16468.653} C_VEL
LIN {X 0,Y 298.827,Z 673.233,A -85,B 0,C 180,E1 -16470,E2 -16470} C_VEL
LIN {X 0,Y 298.964,Z 672.475,A -85,B 0,C 180,E1 -16472.695,E2 -16472.695} C_VEL
LIN {X 0,Y 299.084,Z 671.539,A -85,B 0,C 180,E1 -16474.042,E2 -16474.042} C_VEL
LIN {X 0,Y 299.185,Z 670.235,A -85,B 0,C 180,E1 -16475.391,E2 -16475.391} C_VEL
LIN {X 0,Y 299.84,Z 667.415,A -85,B 0,C 180,E1 -16477.407,E2 -16477.407} C_VEL
LIN {X 0,Y 300.72,Z 663.587,A -85,B 0,C 180,E1 -16479.415,E2 -16479.415} C_VEL
LIN {X 0,Y 301.563,Z 658.506,A -85,B 0,C 180,E1 -16481.493,E2 -16481.493} C_VEL
LIN {X 0,Y 302.712,Z 652.474,A -85,B 0,C 180,E1 -16483.424,E2 -16483.424} C_VEL
LIN {X 0,Y 304.119,Z 644.691,A -85,B 0,C 180,E1 -16485.412,E2 -16485.412} C_VEL
LIN {X 0,Y 305.584,Z 635.018,A -85,B 0,C 180,E1 -16487.396,E2 -16487.396} C_VEL
LIN {X 0,Y 306.901,Z 625.971,A -85,B 0,C 180,E1 -16488.872,E2 -16488.872} C_VEL
LIN {X 0,Y 308.303,Z 615.462,A -85,B 0,C 180,E1 -16490.247,E2 -16490.247} C_VEL
LIN {X 0,Y 309.512,Z 603.78,A -85,B 0,C 180,E1 -16491.46,E2 -16491.46} C_VEL
LIN {X 0,Y 310.502,Z 592.313,A -85,B 0,C 180,E1 -16492.366,E2 -16492.366} C_VEL
LIN {X 0,Y 310.956,Z 579.863,A -85,B 0,C 180,E1 -16493.1,E2 -16493.1} C_VEL
LIN {X 0,Y 311.189,Z 567.02,A -85,B 0,C 180,E1 -16493.588,E2 -16493.588} C_VEL
LIN {X 0,Y 311.682,Z 530.569,A -85,B 0,C 180,E1 -16494.464,E2 -16494.464} C_VEL
LIN {X 0,Y 311.949,Z 516.651,A -85,B 0,C 180,E1 -16494.788,E2 -16494.788} C_VEL
LIN {X 0,Y 303.839,Z 498.706,A -85,B 0,C 180,E1 -16495.993,E2 -16495.993} C_VEL
LIN {X 0,Y 298.647,Z 488.16,A -85,B 0,C 180,E1 -16496.821,E2 -16496.821} C_VEL
LIN {X 0,Y 298.487,Z 487.337,A -85,B 0,C 180,E1 -16497.118,E2 -16497.118} C_VEL
LIN {X 0,Y 298.392,Z 487.31,A -85,B 0,C 180,E1 -16501.208,E2 -16501.208} C_VEL
LIN {X 0,Y 298.427,Z 487.313,A -85,B 0,C 180,E1 -16504.487,E2 -16504.487} C_VEL
LIN {X 0,Y 298.412,Z 487.298,A -85,B 0,C 180,E1 -16507.757,E2 -16507.757} C_VEL
LIN {X 0,Y 298.383,Z 487.303,A -85,B 0,C 180,E1 -16511.261,E2 -16511.261} C_VEL
LIN {X 0,Y 298.386,Z 487.312,A -85,B 0,C 180,E1 -16515.041,E2 -16515.041} C_VEL
LIN {X 0,Y 298.384,Z 487.283,A -85,B 0,C 180,E1 -16518.912,E2 -16518.912} C_VEL
LIN {X 0,Y 298.44,Z 487.305,A -85,B 0,C 180,E1 -16523.192,E2 -16523.192} C_VEL
LIN {X 0,Y 298.391,Z 487.288,A -85,B 0,C 180,E1 -16527.199,E2 -16527.199} C_VEL
LIN {X 0,Y 298.426,Z 487.268,A -85,B 0,C 180,E1 -16530.625,E2 -16530.625} C_VEL
LIN {X 0,Y 297.746,Z 487.371,A -85,B 0,C 180,E1 -16531.751,E2 -16531.751} C_VEL
LIN {X 0,Y 294.909,Z 487.747,A -85,B 0,C 180,E1 -16533.587,E2 -16533.587} C_VEL
LIN {X 0,Y 292.506,Z 488.051,A -85,B 0,C 180,E1 -16535.076,E2 -16535.076} C_VEL
LIN {X 0,Y 291.463,Z 488.174,A -85,B 0,C 180,E1 -16536.228,E2 -16536.228} C_VEL
LIN {X 0,Y 291.371,Z 488.181,A -85,B 0,C 180,E1 -16536.619,E2 -16536.619} C_VEL
LIN {X 0,Y 291.453,Z 488.179,A -85,B 0,C 180,E1 -16540.27,E2 -16540.27} C_VEL
LIN {X 0,Y 291.535,Z 488.156,A -85,B 0,C 180,E1 -16544.634,E2 -16544.634} C_VEL
LIN {X 0,Y 291.53,Z 488.163,A -85,B 0,C 180,E1 -16548.88,E2 -16548.88} C_VEL
LIN {X 0,Y 291.703,Z 488.135,A -85,B 0,C 180,E1 -16551.688,E2 -16551.688} C_VEL
LIN {X 0,Y 291.624,Z 488.155,A -85,B 0,C 180,E1 -16554.468,E2 -16554.468} C_VEL
LIN {X 0,Y 291.884,Z 488.112,A -85,B 0,C 180,E1 -16558.62,E2 -16558.62} C_VEL
LIN {X 0,Y 291.884,Z 488.124,A -85,B 0,C 180,E1 -16561.38,E2 -16561.38} C_VEL
LIN {X 0,Y 291.73,Z 488.142,A -85,B 0,C 180,E1 -16566.918,E2 -16566.918} C_VEL
LIN {X 0,Y 291.568,Z 488.153,A -85,B 0,C 180,E1 -16569.714,E2 -16569.714} C_VEL
LIN {X 0,Y 291.515,Z 488.173,A -85,B 0,C 180,E1 -16573.951,E2 -16573.951} C_VEL
LIN {X 0,Y 291.479,Z 488.16,A -85,B 0,C 180,E1 -16576.818,E2 -16576.818} C_VEL
LIN {X 0,Y 291.445,Z 488.149,A -85,B 0,C 180,E1 -16579.875,E2 -16579.875} C_VEL
LIN {X 0,Y 291.393,Z 488.184,A -85,B 0,C 180,E1 -16584.206,E2 -16584.206} C_VEL
LIN {X 0,Y 291.418,Z 488.158,A -85,B 0,C 180,E1 -16587.272,E2 -16587.272} C_VEL
LIN {X 0,Y 291.333,Z 488.195,A -85,B 0,C 180,E1 -16590.437,E2 -16590.437} C_VEL
LIN {X 0,Y 291.34,Z 488.177,A -85,B 0,C 180,E1 -16593.699,E2 -16593.699} C_VEL
LIN {X 0,Y 291.368,Z 488.183,A -85,B 0,C 180,E1 -16597.254,E2 -16597.254} C_VEL
LIN {X 0,Y 291.329,Z 488.197,A -85,B 0,C 180,E1 -16600.643,E2 -16600.643} C_VEL
LIN {X 0,Y 291.33,Z 488.156,A -85,B 0,C 180,E1 -16604.394,E2 -16604.394} C_VEL
LIN {X 0,Y 291.384,Z 488.171,A -85,B 0,C 180,E1 -16608.392,E2 -16608.392} C_VEL
LIN {X 0,Y 291.459,Z 488.424,A -85,B 0,C 180,E1 -16609.553,E2 -16609.553} C_VEL
LIN {X 0,Y 294.207,Z 498.964,A -85,B 0,C 180,E1 -16612.617,E2 -16612.617} C_VEL
LIN {X 0,Y 296.858,Z 510.056,A -85,B 0,C 180,E1 -16615.622,E2 -16615.622} C_VEL
LIN {X 0,Y 299.047,Z 520.428,A -85,B 0,C 180,E1 -16618.291,E2 -16618.291} C_VEL
LIN {X 0,Y 298.651,Z 524.499,A -85,B 0,C 180,E1 -16619.215,E2 -16619.215} C_VEL
LIN {X 0,Y 296.477,Z 538.815,A -85,B 0,C 180,E1 -16622.373,E2 -16622.373} C_VEL
LIN {X 0,Y 299.906,Z 565.661,A -85,B 0,C 180,E1 -16623.446,E2 -16623.446} C_VEL
LIN {X 0,Y 303.009,Z 596.277,A -85,B 0,C 180,E1 -16624.51,E2 -16624.51} C_VEL
LIN {X 0,Y 303.633,Z 606.667,A -85,B 0,C 180,E1 -16624.828,E2 -16624.828} C_VEL
LIN {X 0,Y 302.411,Z 650.139,A -85,B 0,C 180,E1 -16625.866,E2 -16625.866} C_VEL
LIN {X 0,Y 301.583,Z 663.381,A -85,B 0,C 180,E1 -16626.435,E2 -16626.435} C_VEL
LIN {X 0,Y 300.269,Z 675.544,A -85,B 0,C 180,E1 -16627.192,E2 -16627.192} C_VEL
LIN {X 0,Y 298.619,Z 687.855,A -85,B 0,C 180,E1 -16628.243,E2 -16628.243} C_VEL
LIN {X 0,Y 296.786,Z 699.528,A -85,B 0,C 180,E1 -16629.557,E2 -16629.557} C_VEL
LIN {X 0,Y 295.086,Z 710.085,A -85,B 0,C 180,E1 -16631.065,E2 -16631.065} C_VEL
LIN {X 0,Y 293.633,Z 718.747,A -85,B 0,C 180,E1 -16632.592,E2 -16632.592} C_VEL
LIN {X 0,Y 292.012,Z 727.463,A -85,B 0,C 180,E1 -16634.47,E2 -16634.47} C_VEL
LIN {X 0,Y 291.319,Z 733.463,A -85,B 0,C 180,E1 -16636.04,E2 -16636.04} C_VEL
LIN {X 0,Y 290.594,Z 740.106,A -85,B 0,C 180,E1 -16638.137,E2 -16638.137} C_VEL
LIN {X 0,Y 290.231,Z 745.422,A -85,B 0,C 180,E1 -16640.241,E2 -16640.241} C_VEL
LIN {X 0,Y 290.232,Z 749.595,A -85,B 0,C 180,E1 -16642.347,E2 -16642.347} C_VEL
LIN {X 0,Y 290.443,Z 752.709,A -85,B 0,C 180,E1 -16644.446,E2 -16644.446} C_VEL
LIN {X 0,Y 290.717,Z 754.216,A -85,B 0,C 180,E1 -16645.841,E2 -16645.841} C_VEL
LIN {X 0,Y 291.155,Z 755.964,A -85,B 0,C 180,E1 -16648.617,E2 -16648.617} C_VEL
LIN {X 0,Y 291.449,Z 756.229,A -85,B 0,C 180,E1 -16650,E2 -16650} C_VEL
LIN {X 0,Y 291.157,Z 755.957,A -85,B 0,C 180,E1 -16651.383,E2 -16651.383} C_VEL
LIN {X 0,Y 290.721,Z 754.203,A -85,B 0,C 180,E1 -16654.159,E2 -16654.159} C_VEL
LIN {X 0,Y 290.455,Z 752.689,A -85,B 0,C 180,E1 -16655.554,E2 -16655.554} C_VEL
LIN {X 0,Y 290.271,Z 749.569,A -85,B 0,C 180,E1 -16657.652,E2 -16657.652} C_VEL
LIN {X 0,Y 290.231,Z 745.375,A -85,B 0,C 180,E1 -16659.759,E2 -16659.759} C_VEL
LIN {X 0,Y 290.702,Z 739.011,A -85,B 0,C 180,E1 -16662.212,E2 -16662.212} C_VEL
LIN {X 0,Y 291.547,Z 732.124,A -85,B 0,C 180,E1 -16664.305,E2 -16664.305} C_VEL
LIN {X 0,Y 292.535,Z 725.066,A -85,B 0,C 180,E1 -16666.058,E2 -16666.058} C_VEL
LIN {X 0,Y 293.844,Z 716.801,A -85,B 0,C 180,E1 -16667.755,E2 -16667.755} C_VEL
LIN {X 0,Y 295.546,Z 706.671,A -85,B 0,C 180,E1 -16669.445,E2 -16669.445} C_VEL
LIN {X 0,Y 297.451,Z 695.274,A -85,B 0,C 180,E1 -16670.938,E2 -16670.938} C_VEL
LIN {X 0,Y 299.117,Z 684.14,A -85,B 0,C 180,E1 -16672.081,E2 -16672.081} C_VEL
LIN {X 0,Y 300.701,Z 671.819,A -85,B 0,C 180,E1 -16673.046,E2 -16673.046} C_VEL
LIN {X 0,Y 301.821,Z 658.931,A -85,B 0,C 180,E1 -16673.768,E2 -16673.768} C_VEL
LIN {X 0,Y 302.52,Z 645.39,A -85,B 0,C 180,E1 -16674.25,E2 -16674.25} C_VEL
LIN {X 0,Y 303.547,Z 604.037,A -85,B 0,C 180,E1 -16675.22,E2 -16675.22} C_VEL
LIN {X 0,Y 300.55,Z 571.708,A -85,B 0,C 180,E1 -16676.311,E2 -16676.311} C_VEL
LIN {X 0,Y 296.638,Z 540.842,A -85,B 0,C 180,E1 -16677.484,E2 -16677.484} C_VEL
LIN {X 0,Y 296.436,Z 538.658,A -85,B 0,C 180,E1 -16677.631,E2 -16677.631} C_VEL
LIN {X 0,Y 299.05,Z 521.564,A -85,B 0,C 180,E1 -16681.414,E2 -16681.414} C_VEL
LIN {X 0,Y 297.483,Z 512.939,A -85,B 0,C 180,E1 -16683.589,E2 -16683.589} C_VEL
LIN {X 0,Y 295.432,Z 503.815,A -85,B 0,C 180,E1 -16686.019,E2 -16686.019} C_VEL
LIN {X 0,Y 292.468,Z 492.148,A -85,B 0,C 180,E1 -16689.294,E2 -16689.294} C_VEL
LIN {X 0,Y 291.414,Z 488.291,A -85,B 0,C 180,E1 -16690.491,E2 -16690.491} C_VEL
LIN {X 0,Y 291.35,Z 488.167,A -85,B 0,C 180,E1 -16694.389,E2 -16694.389} C_VEL
LIN {X 0,Y 291.324,Z 488.186,A -85,B 0,C 180,E1 -16698.403,E2 -16698.403} C_VEL
LIN {X 0,Y 291.343,Z 488.182,A -85,B 0,C 180,E1 -16701.157,E2 -16701.157} C_VEL
LIN {X 0,Y 291.357,Z 488.19,A -85,B 0,C 180,E1 -16704.625,E2 -16704.625} C_VEL
LIN {X 0,Y 291.367,Z 488.18,A -85,B 0,C 180,E1 -16707.95,E2 -16707.95} C_VEL
LIN {X 0,Y 291.378,Z 488.183,A -85,B 0,C 180,E1 -16711.158,E2 -16711.158} C_VEL
LIN {X 0,Y 291.41,Z 488.165,A -85,B 0,C 180,E1 -16714.271,E2 -16714.271} C_VEL
LIN {X 0,Y 291.369,Z 488.189,A -85,B 0,C 180,E1 -16717.299,E2 -16717.299} C_VEL
LIN {X 0,Y 291.452,Z 488.147,A -85,B 0,C 180,E1 -16720.27,E2 -16720.27} C_VEL
LIN {X 0,Y 291.549,Z 488.166,A -85,B 0,C 180,E1 -16724.623,E2 -16724.623} C_VEL
LIN {X 0,Y 291.528,Z 488.153,A -85,B 0,C 180,E1 -16728.88,E2 -16728.88} C_VEL
LIN {X 0,Y 291.682,Z 488.15,A -85,B 0,C 180,E1 -16731.688,E2 -16731.688} C_VEL
LIN {X 0,Y 291.623,Z 488.145,A -85,B 0,C 180,E1 -16734.468,E2 -16734.468} C_VEL
LIN {X 0,Y 291.884,Z 488.127,A -85,B 0,C 180,E1 -16738.62,E2 -16738.62} C_VEL
LIN {X 0,Y 291.884,Z 488.115,A -85,B 0,C 180,E1 -16741.38,E2 -16741.38} C_VEL
LIN {X 0,Y 291.731,Z 488.142,A -85,B 0,C 180,E1 -16746.918,E2 -16746.918} C_VEL
LIN {X 0,Y 291.568,Z 488.145,A -85,B 0,C 180,E1 -16749.714,E2 -16749.714} C_VEL
LIN {X 0,Y 291.515,Z 488.17,A -85,B 0,C 180,E1 -16753.951,E2 -16753.951} C_VEL
LIN {X 0,Y 291.48,Z 488.162,A -85,B 0,C 180,E1 -16756.818,E2 -16756.818} C_VEL
LIN {X 0,Y 291.445,Z 488.18,A -85,B 0,C 180,E1 -16759.875,E2 -16759.875} C_VEL
LIN {X 0,Y 291.378,Z 488.185,A -85,B 0,C 180,E1 -16764.207,E2 -16764.207} C_VEL
LIN {X 0,Y 291.418,Z 488.173,A -85,B 0,C 180,E1 -16767.272,E2 -16767.272} C_VEL
LIN {X 0,Y 291.332,Z 488.141,A -85,B 0,C 180,E1 -16770.438,E2 -16770.438} C_VEL
LIN {X 0,Y 291.34,Z 488.178,A -85,B 0,C 180,E1 -16773.699,E2 -16773.699} C_VEL
LIN {X 0,Y 291.368,Z 488.182,A -85,B 0,C 180,E1 -16777.254,E2 -16777.254} C_VEL
LIN {X 0,Y 291.329,Z 488.156,A -85,B 0,C 180,E1 -16780.643,E2 -16780.643} C_VEL
LIN {X 0,Y 291.312,Z 488.199,A -85,B 0,C 180,E1 -16784.398,E2 -16784.398} C_VEL
LIN {X 0,Y 291.325,Z 488.173,A -85,B 0,C 180,E1 -16788.405,E2 -16788.405} C_VEL
LIN {X 0,Y 291.362,Z 488.189,A -85,B 0,C 180,E1 -16791.161,E2 -16791.161} C_VEL
LIN {X 0,Y 291.36,Z 488.119,A -85,B 0,C 180,E1 -16794.627,E2 -16794.627} C_VEL
LIN {X 0,Y 291.371,Z 488.149,A -85,B 0,C 180,E1 -16797.952,E2 -16797.952} C_VEL
LIN {X 0,Y 291.431,Z 488.28,A -85,B 0,C 180,E1 -16802.327,E2 -16802.327} C_VEL
LIN {X 0,Y 291.63,Z 489.232,A -85,B 0,C 180,E1 -16802.617,E2 -16802.617} C_VEL
LIN {X 0,Y 299.529,Z 505.088,A -85,B 0,C 180,E1 -16803.876,E2 -16803.876} C_VEL
LIN {X 0,Y 305.498,Z 518.479,A -85,B 0,C 180,E1 -16804.793,E2 -16804.793} C_VEL
LIN {X 0,Y 304.71,Z 567.65,A -85,B 0,C 180,E1 -16805.987,E2 -16805.987} C_VEL
LIN {X 0,Y 304.422,Z 580.977,A -85,B 0,C 180,E1 -16806.5,E2 -16806.5} C_VEL
LIN {X 0,Y 303.816,Z 592.931,A -85,B 0,C 180,E1 -16807.204,E2 -16807.204} C_VEL
LIN {X 0,Y 302.858,Z 605.181,A -85,B 0,C 180,E1 -16808.205,E2 -16808.205} C_VEL
LIN {X 0,Y 301.756,Z 615.447,A -85,B 0,C 180,E1 -16809.285,E2 -16809.285} C_VEL
LIN {X 0,Y 300.303,Z 626.191,A -85,B 0,C 180,E1 -16810.697,E2 -16810.697} C_VEL
LIN {X 0,Y 298.926,Z 635.387,A -85,B 0,C 180,E1 -16812.204,E2 -16812.204} C_VEL
LIN {X 0,Y 297.623,Z 643.742,A -85,B 0,C 180,E1 -16813.892,E2 -16813.892} C_VEL
LIN {X 0,Y 296.155,Z 651.855,A -85,B 0,C 180,E1 -16815.922,E2 -16815.922} C_VEL
LIN {X 0,Y 294.755,Z 658.964,A -85,B 0,C 180,E1 -16818.164,E2 -16818.164} C_VEL
LIN {X 0,Y 293.814,Z 664.336,A -85,B 0,C 180,E1 -16820.361,E2 -16820.361} C_VEL
LIN {X 0,Y 292.879,Z 668.226,A -85,B 0,C 180,E1 -16822.416,E2 -16822.416} C_VEL
LIN {X 0,Y 292.199,Z 671.094,A -85,B 0,C 180,E1 -16824.479,E2 -16824.479} C_VEL
LIN {X 0,Y 292.078,Z 672.438,A -85,B 0,C 180,E1 -16825.861,E2 -16825.861} C_VEL
LIN {X 0,Y 291.847,Z 673.994,A -85,B 0,C 180,E1 -16828.62,E2 -16828.62} C_VEL
LIN {X 0,Y 291.8,Z 674.221,A -85,B 0,C 180,E1 -16830,E2 -16830} C_VEL
LIN {X 0,Y 291.955,Z 673.461,A -85,B 0,C 180,E1 -16832.759,E2 -16832.759} C_VEL
LIN {X 0,Y 292.072,Z 672.526,A -85,B 0,C 180,E1 -16834.14,E2 -16834.14} C_VEL
LIN {X 0,Y 292.186,Z 671.223,A -85,B 0,C 180,E1 -16835.521,E2 -16835.521} C_VEL
LIN {X 0,Y 292.872,Z 668.402,A -85,B 0,C 180,E1 -16837.584,E2 -16837.584} C_VEL
LIN {X 0,Y 293.789,Z 664.574,A -85,B 0,C 180,E1 -16839.64,E2 -16839.64} C_VEL
LIN {X 0,Y 294.679,Z 659.493,A -85,B 0,C 180,E1 -16841.765,E2 -16841.765} C_VEL
LIN {X 0,Y 295.881,Z 653.461,A -85,B 0,C 180,E1 -16843.74,E2 -16843.74} C_VEL
LIN {X 0,Y 297.35,Z 645.677,A -85,B 0,C 180,E1 -16845.771,E2 -16845.771} C_VEL
LIN {X 0,Y 298.883,Z 636.003,A -85,B 0,C 180,E1 -16847.799,E2 -16847.799} C_VEL
LIN {X 0,Y 300.258,Z 626.956,A -85,B 0,C 180,E1 -16849.306,E2 -16849.306} C_VEL
LIN {X 0,Y 301.728,Z 616.443,A -85,B 0,C 180,E1 -16850.708,E2 -16850.708} C_VEL
LIN {X 0,Y 302.981,Z 604.763,A -85,B 0,C 180,E1 -16851.946,E2 -16851.946} C_VEL
LIN {X 0,Y 304.01,Z 593.294,A -85,B 0,C 180,E1 -16852.871,E2 -16852.871} C_VEL
LIN {X 0,Y 304.484,Z 581.049,A -85,B 0,C 180,E1 -16853.61,E2 -16853.61} C_VEL
LIN {X 0,Y 304.764,Z 567.379,A -85,B 0,C 180,E1 -16854.135,E2 -16854.135} C_VEL
LIN {X 0,Y 305.256,Z 532.299,A -85,B 0,C 180,E1 -16854.994,E2 -16854.994} C_VEL
LIN {X 0,Y 305.535,Z 518.534,A -85,B 0,C 180,E1 -16855.322,E2 -16855.322} C_VEL
LIN {X 0,Y 297.306,Z 500.393,A -85,B 0,C 180,E1 -16856.591,E2 -16856.591} C_VEL
LIN {X 0,Y 291.678,Z 489.28,A -85,B 0,C 180,E1 -16857.497,E2 -16857.497} C_VEL
LIN {X 0,Y 291.453,Z 488.3,A -85,B 0,C 180,E1 -16857.754,E2 -16857.754} C_VEL
LIN {X 0,Y 291.37,Z 488.177,A -85,B 0,C 180,E1 -16862.049,E2 -16862.049} C_VEL
LIN {X 0,Y 291.36,Z 488.186,A -85,B 0,C 180,E1 -16865.373,E2 -16865.373} C_VEL
LIN {X 0,Y 291.351,Z 488.19,A -85,B 0,C 180,E1 -16868.841,E2 -16868.841} C_VEL
LIN {X 0,Y 291.317,Z 488.17,A -85,B 0,C 180,E1 -16872.492,E2 -16872.492} C_VEL
LIN {X 0,Y 291.317,Z 488.199,A -85,B 0,C 180,E1 -16876.363,E2 -16876.363} C_VEL
LIN {X 0,Y 291.375,Z 488.149,A -85,B 0,C 180,E1 -16880.518,E2 -16880.518} C_VEL
LIN {X 0,Y 291.4,Z 488.179,A -85,B 0,C 180,E1 -16882.918,E2 -16882.918} C_VEL
LIN {X 0,Y 291.34,Z 488.18,A -85,B 0,C 180,E1 -16886.301,E2 -16886.301} C_VEL
LIN {X 0,Y 291.382,Z 488.14,A -85,B 0,C 180,E1 -16890.26,E2 -16890.26} C_VEL
LIN {X 0,Y 291.411,Z 488.184,A -85,B 0,C 180,E1 -16894.271,E2 -16894.271} C_VEL
LIN {X 0,Y 291.371,Z 488.181,A -85,B 0,C 180,E1 -16896.619,E2 -16896.619} C_VEL
LIN {X 0,Y 290.698,Z 488.261,A -85,B 0,C 180,E1 -16897.773,E2 -16897.773} C_VEL
LIN {X 0,Y 287.897,Z 488.621,A -85,B 0,C 180,E1 -16899.653,E2 -16899.653} C_VEL
LIN {X 0,Y 285.527,Z 488.919,A -85,B 0,C 180,E1 -16901.179,E2 -16901.179} C_VEL
LIN {X 0,Y 284.504,Z 489.039,A -85,B 0,C 180,E1 -16902.36,E2 -16902.36} C_VEL
LIN {X 0,Y 284.417,Z 489.045,A -85,B 0,C 180,E1 -16902.76,E2 -16902.76} C_VEL
LIN {X 0,Y 284.472,Z 489.045,A -85,B 0,C 180,E1 -16905.697,E2 -16905.697} C_VEL
LIN {X 0,Y 284.56,Z 489.019,A -85,B 0,C 180,E1 -16910.044,E2 -16910.044} C_VEL
LIN {X 0,Y 284.692,Z 489.016,A -85,B 0,C 180,E1 -16912.91,E2 -16912.91} C_VEL
LIN {X 0,Y 284.85,Z 488.988,A -85,B 0,C 180,E1 -16918.586,E2 -16918.586} C_VEL
LIN {X 0,Y 284.85,Z 488.999,A -85,B 0,C 180,E1 -16921.414,E2 -16921.414} C_VEL
LIN {X 0,Y 284.681,Z 489.021,A -85,B 0,C 180,E1 -16927.09,E2 -16927.09} C_VEL
LIN {X 0,Y 284.512,Z 489.03,A -85,B 0,C 180,E1 -16929.957,E2 -16929.957} C_VEL
LIN {X 0,Y 284.475,Z 489.049,A -85,B 0,C 180,E1 -16934.303,E2 -16934.303} C_VEL
LIN {X 0,Y 284.416,Z 489.031,A -85,B 0,C 180,E1 -16937.249,E2 -16937.249} C_VEL
LIN {X 0,Y 284.372,Z 489.034,A -85,B 0,C 180,E1 -16940.243,E2 -16940.243} C_VEL
LIN {X 0,Y 284.362,Z 489.062,A -85,B 0,C 180,E1 -16943.875,E2 -16943.875} C_VEL
LIN {X 0,Y 284.392,Z 489.032,A -85,B 0,C 180,E1 -16947.174,E2 -16947.174} C_VEL
LIN {X 0,Y 284.291,Z 489.068,A -85,B 0,C 180,E1 -16951.275,E2 -16951.275} C_VEL
LIN {X 0,Y 284.337,Z 489.065,A -85,B 0,C 180,E1 -16955.349,E2 -16955.349} C_VEL
LIN {X 0,Y 284.304,Z 489.057,A -85,B 0,C 180,E1 -16958.17,E2 -16958.17} C_VEL
LIN {X 0,Y 284.266,Z 489.053,A -85,B 0,C 180,E1 -16962.125,E2 -16962.125} C_VEL
LIN {X 0,Y 284.315,Z 489.054,A -85,B 0,C 180,E1 -16966.202,E2 -16966.202} C_VEL
LIN {X 0,Y 284.391,Z 489.268,A -85,B 0,C 180,E1 -16968.864,E2 -16968.864} C_VEL
LIN {X 0,Y 287.445,Z 500.778,A -85,B 0,C 180,E1 -16972.321,E2 -16972.321} C_VEL
LIN {X 0,Y 290.091,Z 512.039,A -85,B 0,C 180,E1 -16975.459,E2 -16975.459} C_VEL
LIN {X 0,Y 292.137,Z 521.811,A -85,B 0,C 180,E1 -16978.046,E2 -16978.046} C_VEL
LIN {X 0,Y 291.862,Z 525.11,A -85,B 0,C 180,E1 -16978.822,E2 -16978.822} C_VEL
LIN {X 0,Y 289.838,Z 537.772,A -85,B 0,C 180,E1 -16981.683,E2 -16981.683} C_VEL
LIN {X 0,Y 293.188,Z 563.467,A -85,B 0,C 180,E1 -16982.757,E2 -16982.757} C_VEL
LIN {X 0,Y 296.563,Z 596.81,A -85,B 0,C 180,E1 -16983.955,E2 -16983.955} C_VEL
LIN {X 0,Y 297.163,Z 606.895,A -85,B 0,C 180,E1 -16984.272,E2 -16984.272} C_VEL
LIN {X 0,Y 295.897,Z 649.746,A -85,B 0,C 180,E1 -16985.324,E2 -16985.324} C_VEL
LIN {X 0,Y 295.002,Z 663.239,A -85,B 0,C 180,E1 -16985.928,E2 -16985.928} C_VEL
LIN {X 0,Y 293.6,Z 675.674,A -85,B 0,C 180,E1 -16986.737,E2 -16986.737} C_VEL
LIN {X 0,Y 292.031,Z 686.86,A -85,B 0,C 180,E1 -16987.726,E2 -16987.726} C_VEL
LIN {X 0,Y 290.124,Z 698.53,A -85,B 0,C 180,E1 -16989.066,E2 -16989.066} C_VEL
LIN {X 0,Y 288.275,Z 709.074,A -85,B 0,C 180,E1 -16990.6,E2 -16990.6} C_VEL
LIN {X 0,Y 286.789,Z 717.74,A -85,B 0,C 180,E1 -16992.163,E2 -16992.163} C_VEL
LIN {X 0,Y 285.415,Z 725.299,A -85,B 0,C 180,E1 -16993.808,E2 -16993.808} C_VEL
LIN {X 0,Y 284.394,Z 732.461,A -85,B 0,C 180,E1 -16995.693,E2 -16995.693} C_VEL
LIN {X 0,Y 283.593,Z 739.101,A -85,B 0,C 180,E1 -16997.84,E2 -16997.84} C_VEL
LIN {X 0,Y 283.182,Z 744.417,A -85,B 0,C 180,E1 -16999.996,E2 -16999.996} C_VEL
LIN {X 0,Y 283.168,Z 748.593,A -85,B 0,C 180,E1 -17002.155,E2 -17002.155} C_VEL
LIN {X 0,Y 283.352,Z 751.707,A -85,B 0,C 180,E1 -17004.306,E2 -17004.306} C_VEL
LIN {X 0,Y 283.632,Z 753.218,A -85,B 0,C 180,E1 -17005.737,E2 -17005.737} C_VEL
LIN {X 0,Y 284.098,Z 754.972,A -85,B 0,C 180,E1 -17008.583,E2 -17008.583} C_VEL
LIN {X 0,Y 284.416,Z 755.24,A -85,B 0,C 180,E1 -17010,E2 -17010} C_VEL
LIN {X 0,Y 284.1,Z 754.965,A -85,B 0,C 180,E1 -17011.417,E2 -17011.417} C_VEL
LIN {X 0,Y 283.637,Z 753.204,A -85,B 0,C 180,E1 -17014.263,E2 -17014.263} C_VEL
LIN {X 0,Y 283.373,Z 751.688,A -85,B 0,C 180,E1 -17015.693,E2 -17015.693} C_VEL
LIN {X 0,Y 283.186,Z 748.562,A -85,B 0,C 180,E1 -17017.845,E2 -17017.845} C_VEL
LIN {X 0,Y 283.182,Z 744.368,A -85,B 0,C 180,E1 -17020.004,E2 -17020.004} C_VEL
LIN {X 0,Y 283.707,Z 738.003,A -85,B 0,C 180,E1 -17022.518,E2 -17022.518} C_VEL
LIN {X 0,Y 284.633,Z 731.118,A -85,B 0,C 180,E1 -17024.66,E2 -17024.66} C_VEL
LIN {X 0,Y 285.717,Z 723.949,A -85,B 0,C 180,E1 -17026.479,E2 -17026.479} C_VEL
LIN {X 0,Y 287.354,Z 713.955,A -85,B 0,C 180,E1 -17028.538,E2 -17028.538} C_VEL
LIN {X 0,Y 289.294,Z 703.324,A -85,B 0,C 180,E1 -17030.254,E2 -17030.254} C_VEL
LIN {X 0,Y 291.261,Z 691.385,A -85,B 0,C 180,E1 -17031.776,E2 -17031.776} C_VEL
LIN {X 0,Y 293.1,Z 679.406,A -85,B 0,C 180,E1 -17032.932,E2 -17032.932} C_VEL
LIN {X 0,Y 294.594,Z 666.955,A -85,B 0,C 180,E1 -17033.832,E2 -17033.832} C_VEL
LIN {X 0,Y 295.64,Z 653.818,A -85,B 0,C 180,E1 -17034.503,E2 -17034.503} C_VEL
LIN {X 0,Y 296.208,Z 639.155,A -85,B 0,C 180,E1 -17034.944,E2 -17034.944} C_VEL
LIN {X 0,Y 297.058,Z 604.37,A -85,B 0,C 180,E1 -17035.775,E2 -17035.775} C_VEL
LIN {X 0,Y 294.089,Z 572.192,A -85,B 0,C 180,E1 -17036.895,E2 -17036.895} C_VEL
LIN {X 0,Y 290.488,Z 543.217,A -85,B 0,C 180,E1 -17038.025,E2 -17038.025} C_VEL
LIN {X 0,Y 289.791,Z 537.939,A -85,B 0,C 180,E1 -17038.271,E2 -17038.271} C_VEL
LIN {X 0,Y 292.117,Z 523.352,A -85,B 0,C 180,E1 -17041.552,E2 -17041.552} C_VEL
LIN {X 0,Y 291.649,Z 519.62,A -85,B 0,C 180,E1 -17042.498,E2 -17042.498} C_VEL
LIN {X 0,Y 289.141,Z 507.702,A -85,B 0,C 180,E1 -17045.686,E2 -17045.686} C_VEL
LIN {X 0,Y 286.01,Z 495.192,A -85,B 0,C 180,E1 -17049.283,E2 -17049.283} C_VEL
LIN {X 0,Y 284.365,Z 489.165,A -85,B 0,C 180,E1 -17051.182,E2 -17051.182} C_VEL
LIN {X 0,Y 284.305,Z 489.046,A -85,B 0,C 180,E1 -17054.202,E2 -17054.202} C_VEL
LIN {X 0,Y 284.269,Z 489.058,A -85,B 0,C 180,E1 -17058.124,E2 -17058.124} C_VEL
LIN {X 0,Y 284.315,Z 489.057,A -85,B 0,C 180,E1 -17062.278,E2 -17062.278} C_VEL
LIN {X 0,Y 284.304,Z 489.062,A -85,B 0,C 180,E1 -17065.35,E2 -17065.35} C_VEL
LIN {X 0,Y 284.291,Z 489.069,A -85,B 0,C 180,E1 -17068.725,E2 -17068.725} C_VEL
LIN {X 0,Y 284.392,Z 489.033,A -85,B 0,C 180,E1 -17072.826,E2 -17072.826} C_VEL
LIN {X 0,Y 284.357,Z 489.065,A -85,B 0,C 180,E1 -17076.706,E2 -17076.706} C_VEL
LIN {X 0,Y 284.392,Z 489.022,A -85,B 0,C 180,E1 -17081.261,E2 -17081.261} C_VEL
LIN {X 0,Y 284.486,Z 489.044,A -85,B 0,C 180,E1 -17084.459,E2 -17084.459} C_VEL
LIN {X 0,Y 284.481,Z 489.031,A -85,B 0,C 180,E1 -17088.601,E2 -17088.601} C_VEL
LIN {X 0,Y 284.633,Z 489.028,A -85,B 0,C 180,E1 -17091.48,E2 -17091.48} C_VEL
LIN {X 0,Y 284.593,Z 489.022,A -85,B 0,C 180,E1 -17094.331,E2 -17094.331} C_VEL
LIN {X 0,Y 284.85,Z 489.003,A -85,B 0,C 180,E1 -17098.586,E2 -17098.586} C_VEL
LIN {X 0,Y 284.85,Z 488.991,A -85,B 0,C 180,E1 -17101.414,E2 -17101.414} C_VEL
LIN {X 0,Y 284.682,Z 489.019,A -85,B 0,C 180,E1 -17107.091,E2 -17107.091} C_VEL
LIN {X 0,Y 284.513,Z 489.025,A -85,B 0,C 180,E1 -17109.957,E2 -17109.957} C_VEL
LIN {X 0,Y 284.472,Z 489.044,A -85,B 0,C 180,E1 -17114.303,E2 -17114.303} C_VEL
LIN {X 0,Y 284.417,Z 489.045,A -85,B 0,C 180,E1 -17117.249,E2 -17117.249} C_VEL
LIN {X 0,Y 284.372,Z 489.062,A -85,B 0,C 180,E1 -17120.243,E2 -17120.243} C_VEL
LIN {X 0,Y 284.334,Z 489.067,A -85,B 0,C 180,E1 -17124.847,E2 -17124.847} C_VEL
LIN {X 0,Y 284.327,Z 489.044,A -85,B 0,C 180,E1 -17128.011,E2 -17128.011} C_VEL
LIN {X 0,Y 284.29,Z 489.018,A -85,B 0,C 180,E1 -17131.275,E2 -17131.275} C_VEL
LIN {X 0,Y 284.337,Z 489.068,A -85,B 0,C 180,E1 -17135.349,E2 -17135.349} C_VEL
LIN {X 0,Y 284.304,Z 489.046,A -85,B 0,C 180,E1 -17138.17,E2 -17138.17} C_VEL
LIN {X 0,Y 284.266,Z 489.056,A -85,B 0,C 180,E1 -17142.125,E2 -17142.125} C_VEL
LIN {X 0,Y 284.266,Z 489.054,A -85,B 0,C 180,E1 -17146.193,E2 -17146.193} C_VEL
LIN {X 0,Y 284.305,Z 489.071,A -85,B 0,C 180,E1 -17150.025,E2 -17150.025} C_VEL
LIN {X 0,Y 284.333,Z 489.007,A -85,B 0,C 180,E1 -17153.615,E2 -17153.615} C_VEL
LIN {X 0,Y 284.307,Z 489.009,A -85,B 0,C 180,E1 -17157.19,E2 -17157.19} C_VEL
LIN {X 0,Y 284.373,Z 489.174,A -85,B 0,C 180,E1 -17161.593,E2 -17161.593} C_VEL
LIN {X 0,Y 284.63,Z 490.172,A -85,B 0,C 180,E1 -17161.882,E2 -17161.882} C_VEL
LIN {X 0,Y 293.021,Z 506.796,A -85,B 0,C 180,E1 -17163.268,E2 -17163.268} C_VEL
LIN {X 0,Y 299.092,Z 520.311,A -85,B 0,C 180,E1 -17164.235,E2 -17164.235} C_VEL
LIN {X 0,Y 298.305,Z 568.254,A -85,B 0,C 180,E1 -17165.425,E2 -17165.425} C_VEL
LIN {X 0,Y 298.007,Z 581.469,A -85,B 0,C 180,E1 -17165.936,E2 -17165.936} C_VEL
LIN {X 0,Y 297.342,Z 593.929,A -85,B 0,C 180,E1 -17166.679,E2 -17166.679} C_VEL
LIN {X 0,Y 296.344,Z 606.175,A -85,B 0,C 180,E1 -17167.701,E2 -17167.701} C_VEL
LIN {X 0,Y 295.193,Z 616.44,A -85,B 0,C 180,E1 -17168.802,E2 -17168.802} C_VEL
LIN {X 0,Y 293.678,Z 627.183,A -85,B 0,C 180,E1 -17170.244,E2 -17170.244} C_VEL
LIN {X 0,Y 292.241,Z 636.378,A -85,B 0,C 180,E1 -17171.783,E2 -17171.783} C_VEL
LIN {X 0,Y 290.877,Z 644.733,A -85,B 0,C 180,E1 -17173.508,E2 -17173.508} C_VEL
LIN {X 0,Y 289.343,Z 652.845,A -85,B 0,C 180,E1 -17175.584,E2 -17175.584} C_VEL
LIN {X 0,Y 287.88,Z 659.953,A -85,B 0,C 180,E1 -17177.877,E2 -17177.877} C_VEL
LIN {X 0,Y 286.888,Z 665.325,A -85,B 0,C 180,E1 -17180.126,E2 -17180.126} C_VEL
LIN {X 0,Y 285.914,Z 669.216,A -85,B 0,C 180,E1 -17182.23,E2 -17182.23} C_VEL
LIN {X 0,Y 285.202,Z 672.084,A -85,B 0,C 180,E1 -17184.343,E2 -17184.343} C_VEL
LIN {X 0,Y 285.067,Z 673.427,A -85,B 0,C 180,E1 -17185.759,E2 -17185.759} C_VEL
LIN {X 0,Y 284.955,Z 674.384,A -85,B 0,C 180,E1 -17187.173,E2 -17187.173} C_VEL
LIN {X 0,Y 284.773,Z 675.209,A -85,B 0,C 180,E1 -17190,E2 -17190} C_VEL
LIN {X 0,Y 284.945,Z 674.447,A -85,B 0,C 180,E1 -17192.827,E2 -17192.827} C_VEL
LIN {X 0,Y 285.189,Z 672.211,A -85,B 0,C 180,E1 -17195.657,E2 -17195.657} C_VEL
LIN {X 0,Y 285.907,Z 669.389,A -85,B 0,C 180,E1 -17197.77,E2 -17197.77} C_VEL
LIN {X 0,Y 286.862,Z 665.56,A -85,B 0,C 180,E1 -17199.875,E2 -17199.875} C_VEL
LIN {X 0,Y 287.802,Z 660.48,A -85,B 0,C 180,E1 -17202.05,E2 -17202.05} C_VEL
LIN {X 0,Y 289.058,Z 654.447,A -85,B 0,C 180,E1 -17204.071,E2 -17204.071} C_VEL
LIN {X 0,Y 290.592,Z 646.663,A -85,B 0,C 180,E1 -17206.148,E2 -17206.148} C_VEL
LIN {X 0,Y 292.198,Z 636.988,A -85,B 0,C 180,E1 -17208.22,E2 -17208.22} C_VEL
LIN {X 0,Y 293.635,Z 627.94,A -85,B 0,C 180,E1 -17209.759,E2 -17209.759} C_VEL
LIN {X 0,Y 295.164,Z 617.426,A -85,B 0,C 180,E1 -17211.19,E2 -17211.19} C_VEL
LIN {X 0,Y 296.445,Z 605.902,A -85,B 0,C 180,E1 -17212.44,E2 -17212.44} C_VEL
LIN {X 0,Y 297.533,Z 594.613,A -85,B 0,C 180,E1 -17213.37,E2 -17213.37} C_VEL
LIN {X 0,Y 298.038,Z 582.249,A -85,B 0,C 180,E1 -17214.142,E2 -17214.142} C_VEL
LIN {X 0,Y 298.312,Z 569.115,A -85,B 0,C 180,E1 -17214.668,E2 -17214.668} C_VEL
LIN {X 0,Y 298.925,Z 531.087,A -85,B 0,C 180,E1 -17215.618,E2 -17215.618} C_VEL
LIN {X 0,Y 299.145,Z 520.474,A -85,B 0,C 180,E1 -17215.877,E2 -17215.877} C_VEL
LIN {X 0,Y 291.282,Z 503.109,A -85,B 0,C 180,E1 -17217.136,E2 -17217.136} C_VEL
LIN {X 0,Y 284.562,Z 490.077,A -85,B 0,C 180,E1 -17218.258,E2 -17218.258} C_VEL
LIN {X 0,Y 284.363,Z 489.136,A -85,B 0,C 180,E1 -17218.559,E2 -17218.559} C_VEL
LIN {X 0,Y 284.305,Z 489.057,A -85,B 0,C 180,E1 -17222.944,E2 -17222.944} C_VEL
LIN {X 0,Y 284.331,Z 489.049,A -85,B 0,C 180,E1 -17226.385,E2 -17226.385} C_VEL
LIN {X 0,Y 284.304,Z 489.072,A -85,B 0,C 180,E1 -17229.994,E2 -17229.994} C_VEL
LIN {X 0,Y 284.263,Z 489.06,A -85,B 0,C 180,E1 -17234.194,E2 -17234.194} C_VEL
LIN {X 0,Y 284.269,Z 489.053,A -85,B 0,C 180,E1 -17238.124,E2 -17238.124} C_VEL
LIN {X 0,Y 284.304,Z 489.044,A -85,B 0,C 180,E1 -17241.83,E2 -17241.83} C_VEL
LIN {X 0,Y 284.304,Z 489.066,A -85,B 0,C 180,E1 -17245.35,E2 -17245.35} C_VEL
LIN {X 0,Y 284.29,Z 489.019,A -85,B 0,C 180,E1 -17248.725,E2 -17248.725} C_VEL
LIN {X 0,Y 284.393,Z 489.048,A -85,B 0,C 180,E1 -17252.826,E2 -17252.826} C_VEL
LIN {X 0,Y 284.328,Z 489.057,A -85,B 0,C 180,E1 -17256.703,E2 -17256.703} C_VEL
LIN {X 0,Y 284.393,Z 489.059,A -85,B 0,C 180,E1 -17261.261,E2 -17261.261} C_VEL
LIN {X 0,Y 284.417,Z 489.045,A -85,B 0,C 180,E1 -17262.76,E2 -17262.76} C_VEL
LIN {X 0,Y 283.735,Z 489.126,A -85,B 0,C 180,E1 -17263.943,E2 -17263.943} C_VEL
LIN {X 0,Y 280.881,Z 489.495,A -85,B 0,C 180,E1 -17265.871,E2 -17265.871} C_VEL
LIN {X 0,Y 278.493,Z 489.795,A -85,B 0,C 180,E1 -17267.436,E2 -17267.436} C_VEL
LIN {X 0,Y 277.504,Z 489.913,A -85,B 0,C 180,E1 -17268.649,E2 -17268.649} C_VEL
LIN {X 0,Y 277.442,Z 489.911,A -85,B 0,C 180,E1 -17269.059,E2 -17269.059} C_VEL
LIN {X 0,Y 277.61,Z 489.885,A -85,B 0,C 180,E1 -17271.263,E2 -17271.263} C_VEL
LIN {X 0,Y 277.566,Z 489.906,A -85,B 0,C 180,E1 -17274.187,E2 -17274.187} C_VEL
LIN {X 0,Y 277.816,Z 489.864,A -85,B 0,C 180,E1 -17278.55,E2 -17278.55} C_VEL
LIN {X 0,Y 277.816,Z 489.875,A -85,B 0,C 180,E1 -17281.45,E2 -17281.45} C_VEL
LIN {X 0,Y 277.635,Z 489.9,A -85,B 0,C 180,E1 -17287.271,E2 -17287.271} C_VEL
LIN {X 0,Y 277.455,Z 489.907,A -85,B 0,C 180,E1 -17290.213,E2 -17290.213} C_VEL
LIN {X 0,Y 277.428,Z 489.926,A -85,B 0,C 180,E1 -17294.674,E2 -17294.674} C_VEL
LIN {X 0,Y 277.336,Z 489.9,A -85,B 0,C 180,E1 -17299.234,E2 -17299.234} C_VEL
LIN {X 0,Y 277.312,Z 489.938,A -85,B 0,C 180,E1 -17304.17,E2 -17304.17} C_VEL
LIN {X 0,Y 277.321,Z 489.914,A -85,B 0,C 180,E1 -17307.506,E2 -17307.506} C_VEL
LIN {X 0,Y 277.268,Z 489.947,A -85,B 0,C 180,E1 -17310.482,E2 -17310.482} C_VEL
LIN {X 0,Y 277.243,Z 489.933,A -85,B 0,C 180,E1 -17313.896,E2 -17313.896} C_VEL
LIN {X 0,Y 277.26,Z 489.937,A -85,B 0,C 180,E1 -17317.471,E2 -17317.471} C_VEL
LIN {X 0,Y 277.206,Z 489.949,A -85,B 0,C 180,E1 -17321.237,E2 -17321.237} C_VEL
LIN {X 0,Y 277.24,Z 489.916,A -85,B 0,C 180,E1 -17325.218,E2 -17325.218} C_VEL
LIN {X 0,Y 277.34,Z 490.084,A -85,B 0,C 180,E1 -17328.119,E2 -17328.119} C_VEL
LIN {X 0,Y 280.305,Z 501.139,A -85,B 0,C 180,E1 -17331.583,E2 -17331.583} C_VEL
LIN {X 0,Y 283.27,Z 513.701,A -85,B 0,C 180,E1 -17335.206,E2 -17335.206} C_VEL
LIN {X 0,Y 285.283,Z 524.077,A -85,B 0,C 180,E1 -17338.019,E2 -17338.019} C_VEL
LIN {X 0,Y 283.23,Z 536.903,A -85,B 0,C 180,E1 -17340.98,E2 -17340.98} C_VEL
LIN {X 0,Y 286.937,Z 565.37,A -85,B 0,C 180,E1 -17342.191,E2 -17342.191} C_VEL
LIN {X 0,Y 290.172,Z 597.735,A -85,B 0,C 180,E1 -17343.388,E2 -17343.388} C_VEL
LIN {X 0,Y 290.746,Z 607.1,A -85,B 0,C 180,E1 -17343.693,E2 -17343.693} C_VEL
LIN {X 0,Y 289.456,Z 648.404,A -85,B 0,C 180,E1 -17344.722,E2 -17344.722} C_VEL
LIN {X 0,Y 288.504,Z 662.348,A -85,B 0,C 180,E1 -17345.356,E2 -17345.356} C_VEL
LIN {X 0,Y 287.112,Z 674.686,A -85,B 0,C 180,E1 -17346.179,E2 -17346.179} C_VEL
LIN {X 0,Y 285.46,Z 685.865,A -85,B 0,C 180,E1 -17347.185,E2 -17347.185} C_VEL
LIN {X 0,Y 283.434,Z 697.525,A -85,B 0,C 180,E1 -17348.547,E2 -17348.547} C_VEL
LIN {X 0,Y 281.6,Z 708.081,A -85,B 0,C 180,E1 -17350.121,E2 -17350.121} C_VEL
LIN {X 0,Y 279.958,Z 716.732,A -85,B 0,C 180,E1 -17351.712,E2 -17351.712} C_VEL
LIN {X 0,Y 278.472,Z 724.905,A -85,B 0,C 180,E1 -17353.544,E2 -17353.544} C_VEL
LIN {X 0,Y 277.252,Z 732.647,A -85,B 0,C 180,E1 -17355.691,E2 -17355.691} C_VEL
LIN {X 0,Y 276.363,Z 739.98,A -85,B 0,C 180,E1 -17358.262,E2 -17358.262} C_VEL
LIN {X 0,Y 276.085,Z 744.914,A -85,B 0,C 180,E1 -17360.476,E2 -17360.476} C_VEL
LIN {X 0,Y 276.163,Z 749.169,A -85,B 0,C 180,E1 -17362.98,E2 -17362.98} C_VEL
LIN {X 0,Y 276.55,Z 752.22,A -85,B 0,C 180,E1 -17365.628,E2 -17365.628} C_VEL
LIN {X 0,Y 277.04,Z 753.979,A -85,B 0,C 180,E1 -17368.546,E2 -17368.546} C_VEL
LIN {X 0,Y 277.381,Z 754.251,A -85,B 0,C 180,E1 -17370,E2 -17370} C_VEL
LIN {X 0,Y 277.042,Z 753.972,A -85,B 0,C 180,E1 -17371.454,E2 -17371.454} C_VEL
LIN {X 0,Y 276.556,Z 752.205,A -85,B 0,C 180,E1 -17374.372,E2 -17374.372} C_VEL
LIN {X 0,Y 276.206,Z 749.034,A -85,B 0,C 180,E1 -17377.093,E2 -17377.093} C_VEL
LIN {X 0,Y 276.085,Z 744.864,A -85,B 0,C 180,E1 -17379.524,E2 -17379.524} C_VEL
LIN {X 0,Y 276.368,Z 739.917,A -85,B 0,C 180,E1 -17381.738,E2 -17381.738} C_VEL
LIN {X 0,Y 277.254,Z 732.569,A -85,B 0,C 180,E1 -17384.309,E2 -17384.309} C_VEL
LIN {X 0,Y 278.518,Z 724.665,A -85,B 0,C 180,E1 -17386.488,E2 -17386.488} C_VEL
LIN {X 0,Y 279.929,Z 716.599,A -85,B 0,C 180,E1 -17388.29,E2 -17388.29} C_VEL
LIN {X 0,Y 281.714,Z 706.827,A -85,B 0,C 180,E1 -17390.061,E2 -17390.061} C_VEL
LIN {X 0,Y 283.707,Z 696.037,A -85,B 0,C 180,E1 -17391.622,E2 -17391.622} C_VEL
LIN {X 0,Y 285.456,Z 685.63,A -85,B 0,C 180,E1 -17392.815,E2 -17392.815} C_VEL
LIN {X 0,Y 287.263,Z 673.216,A -85,B 0,C 180,E1 -17393.904,E2 -17393.904} C_VEL
LIN {X 0,Y 288.632,Z 659.815,A -85,B 0,C 180,E1 -17394.761,E2 -17394.761} C_VEL
LIN {X 0,Y 289.506,Z 647.033,A -85,B 0,C 180,E1 -17395.298,E2 -17395.298} C_VEL
LIN {X 0,Y 290.625,Z 605.187,A -85,B 0,C 180,E1 -17396.34,E2 -17396.34} C_VEL
LIN {X 0,Y 287.783,Z 573.513,A -85,B 0,C 180,E1 -17397.47,E2 -17397.47} C_VEL
LIN {X 0,Y 284.172,Z 544.112,A -85,B 0,C 180,E1 -17398.651,E2 -17398.651} C_VEL
LIN {X 0,Y 283.209,Z 536.811,A -85,B 0,C 180,E1 -17398.999,E2 -17398.999} C_VEL
LIN {X 0,Y 285.252,Z 523.943,A -85,B 0,C 180,E1 -17401.985,E2 -17401.985} C_VEL
LIN {X 0,Y 283.591,Z 515.282,A -85,B 0,C 180,E1 -17404.317,E2 -17404.317} C_VEL
LIN {X 0,Y 281.063,Z 504.278,A -85,B 0,C 180,E1 -17407.447,E2 -17407.447} C_VEL
LIN {X 0,Y 278.254,Z 493.474,A -85,B 0,C 180,E1 -17410.736,E2 -17410.736} C_VEL
LIN {X 0,Y 277.312,Z 490.019,A -85,B 0,C 180,E1 -17411.891,E2 -17411.891} C_VEL
LIN {X 0,Y 277.233,Z 489.912,A -85,B 0,C 180,E1 -17415.218,E2 -17415.218} C_VEL
LIN {X 0,Y 277.22,Z 489.954,A -85,B 0,C 180,E1 -17419.511,E2 -17419.511} C_VEL
LIN {X 0,Y 277.26,Z 489.937,A -85,B 0,C 180,E1 -17422.529,E2 -17422.529} C_VEL
LIN {X 0,Y 277.243,Z 489.933,A -85,B 0,C 180,E1 -17426.104,E2 -17426.104} C_VEL
LIN {X 0,Y 277.257,Z 489.949,A -85,B 0,C 180,E1 -17429.538,E2 -17429.538} C_VEL
LIN {X 0,Y 277.354,Z 489.909,A -85,B 0,C 180,E1 -17432.864,E2 -17432.864} C_VEL
LIN {X 0,Y 277.321,Z 489.938,A -85,B 0,C 180,E1 -17436.079,E2 -17436.079} C_VEL
LIN {X 0,Y 277.336,Z 489.901,A -85,B 0,C 180,E1 -17440.766,E2 -17440.766} C_VEL
LIN {X 0,Y 277.428,Z 489.926,A -85,B 0,C 180,E1 -17445.326,E2 -17445.326} C_VEL
LIN {X 0,Y 277.455,Z 489.909,A -85,B 0,C 180,E1 -17449.787,E2 -17449.787} C_VEL
LIN {X 0,Y 277.635,Z 489.901,A -85,B 0,C 180,E1 -17452.729,E2 -17452.729} C_VEL
LIN {X 0,Y 277.816,Z 489.878,A -85,B 0,C 180,E1 -17458.55,E2 -17458.55} C_VEL
LIN {X 0,Y 277.816,Z 489.866,A -85,B 0,C 180,E1 -17461.45,E2 -17461.45} C_VEL
LIN {X 0,Y 277.636,Z 489.895,A -85,B 0,C 180,E1 -17467.271,E2 -17467.271} C_VEL
LIN {X 0,Y 277.455,Z 489.905,A -85,B 0,C 180,E1 -17470.213,E2 -17470.213} C_VEL
LIN {X 0,Y 277.422,Z 489.917,A -85,B 0,C 180,E1 -17474.675,E2 -17474.675} C_VEL
LIN {X 0,Y 277.337,Z 489.939,A -85,B 0,C 180,E1 -17479.235,E2 -17479.235} C_VEL
LIN {X 0,Y 277.287,Z 489.94,A -85,B 0,C 180,E1 -17484.158,E2 -17484.158} C_VEL
LIN {X 0,Y 277.321,Z 489.927,A -85,B 0,C 180,E1 -17487.506,E2 -17487.506} C_VEL
LIN {X 0,Y 277.268,Z 489.891,A -85,B 0,C 180,E1 -17490.482,E2 -17490.482} C_VEL
LIN {X 0,Y 277.243,Z 489.936,A -85,B 0,C 180,E1 -17493.897,E2 -17493.897} C_VEL
LIN {X 0,Y 277.261,Z 489.938,A -85,B 0,C 180,E1 -17497.471,E2 -17497.471} C_VEL
LIN {X 0,Y 277.206,Z 489.919,A -85,B 0,C 180,E1 -17501.237,E2 -17501.237} C_VEL
LIN {X 0,Y 277.215,Z 489.946,A -85,B 0,C 180,E1 -17505.224,E2 -17505.224} C_VEL
LIN {X 0,Y 277.221,Z 489.945,A -85,B 0,C 180,E1 -17509.513,E2 -17509.513} C_VEL
LIN {X 0,Y 277.27,Z 489.911,A -85,B 0,C 180,E1 -17512.532,E2 -17512.532} C_VEL
LIN {X 0,Y 277.246,Z 489.872,A -85,B 0,C 180,E1 -17516.105,E2 -17516.105} C_VEL
LIN {X 0,Y 277.342,Z 490.141,A -85,B 0,C 180,E1 -17520.857,E2 -17520.857} C_VEL
LIN {X 0,Y 277.537,Z 491.046,A -85,B 0,C 180,E1 -17521.089,E2 -17521.089} C_VEL
LIN {X 0,Y 286.589,Z 508.61,A -85,B 0,C 180,E1 -17522.64,E2 -17522.64} C_VEL
LIN {X 0,Y 292.76,Z 522.36,A -85,B 0,C 180,E1 -17523.663,E2 -17523.663} C_VEL
LIN {X 0,Y 291.934,Z 567.597,A -85,B 0,C 180,E1 -17524.801,E2 -17524.801} C_VEL
LIN {X 0,Y 291.661,Z 580.592,A -85,B 0,C 180,E1 -17525.28,E2 -17525.28} C_VEL
LIN {X 0,Y 290.967,Z 593.65,A -85,B 0,C 180,E1 -17526.042,E2 -17526.042} C_VEL
LIN {X 0,Y 290.01,Z 605.952,A -85,B 0,C 180,E1 -17527.056,E2 -17527.056} C_VEL
LIN {X 0,Y 288.652,Z 617.433,A -85,B 0,C 180,E1 -17528.298,E2 -17528.298} C_VEL
LIN {X 0,Y 287.073,Z 628.176,A -85,B 0,C 180,E1 -17529.77,E2 -17529.77} C_VEL
LIN {X 0,Y 285.573,Z 637.37,A -85,B 0,C 180,E1 -17531.342,E2 -17531.342} C_VEL
LIN {X 0,Y 284.145,Z 645.723,A -85,B 0,C 180,E1 -17533.105,E2 -17533.105} C_VEL
LIN {X 0,Y 282.542,Z 653.835,A -85,B 0,C 180,E1 -17535.229,E2 -17535.229} C_VEL
LIN {X 0,Y 281.013,Z 660.943,A -85,B 0,C 180,E1 -17537.576,E2 -17537.576} C_VEL
LIN {X 0,Y 279.966,Z 666.315,A -85,B 0,C 180,E1 -17539.88,E2 -17539.88} C_VEL
LIN {X 0,Y 278.952,Z 670.205,A -85,B 0,C 180,E1 -17542.035,E2 -17542.035} C_VEL
LIN {X 0,Y 278.207,Z 673.073,A -85,B 0,C 180,E1 -17544.201,E2 -17544.201} C_VEL
LIN {X 0,Y 278.058,Z 674.416,A -85,B 0,C 180,E1 -17545.651,E2 -17545.651} C_VEL
LIN {X 0,Y 277.943,Z 675.371,A -85,B 0,C 180,E1 -17547.101,E2 -17547.101} C_VEL
LIN {X 0,Y 277.746,Z 676.198,A -85,B 0,C 180,E1 -17550,E2 -17550} C_VEL
LIN {X 0,Y 277.934,Z 675.434,A -85,B 0,C 180,E1 -17552.899,E2 -17552.899} C_VEL
LIN {X 0,Y 278.193,Z 673.199,A -85,B 0,C 180,E1 -17555.8,E2 -17555.8} C_VEL
LIN {X 0,Y 278.946,Z 670.377,A -85,B 0,C 180,E1 -17557.965,E2 -17557.965} C_VEL
LIN {X 0,Y 279.941,Z 666.547,A -85,B 0,C 180,E1 -17560.121,E2 -17560.121} C_VEL
LIN {X 0,Y 280.933,Z 661.466,A -85,B 0,C 180,E1 -17562.35,E2 -17562.35} C_VEL
LIN {X 0,Y 282.246,Z 655.433,A -85,B 0,C 180,E1 -17564.418,E2 -17564.418} C_VEL
LIN {X 0,Y 283.848,Z 647.648,A -85,B 0,C 180,E1 -17566.543,E2 -17566.543} C_VEL
LIN {X 0,Y 285.53,Z 637.973,A -85,B 0,C 180,E1 -17568.661,E2 -17568.661} C_VEL
LIN {X 0,Y 287.029,Z 628.924,A -85,B 0,C 180,E1 -17570.233,E2 -17570.233} C_VEL
LIN {X 0,Y 288.614,Z 618.412,A -85,B 0,C 180,E1 -17571.695,E2 -17571.695} C_VEL
LIN {X 0,Y 289.991,Z 606.727,A -85,B 0,C 180,E1 -17572.984,E2 -17572.984} C_VEL
LIN {X 0,Y 291.124,Z 595.252,A -85,B 0,C 180,E1 -17573.945,E2 -17573.945} C_VEL
LIN {X 0,Y 291.65,Z 582.694,A -85,B 0,C 180,E1 -17574.733,E2 -17574.733} C_VEL
LIN {X 0,Y 291.932,Z 569.598,A -85,B 0,C 180,E1 -17575.26,E2 -17575.26} C_VEL
LIN {X 0,Y 292.642,Z 529.628,A -85,B 0,C 180,E1 -17576.275,E2 -17576.275} C_VEL
LIN {X 0,Y 292.784,Z 522.408,A -85,B 0,C 180,E1 -17576.456,E2 -17576.456} C_VEL
LIN {X 0,Y 285.179,Z 505.636,A -85,B 0,C 180,E1 -17577.722,E2 -17577.722} C_VEL
LIN {X 0,Y 277.499,Z 490.947,A -85,B 0,C 180,E1 -17579.054,E2 -17579.054} C_VEL
LIN {X 0,Y 277.326,Z 490.023,A -85,B 0,C 180,E1 -17579.37,E2 -17579.37} C_VEL
LIN {X 0,Y 277.246,Z 489.946,A -85,B 0,C 180,E1 -17583.895,E2 -17583.895} C_VEL
LIN {X 0,Y 277.266,Z 489.929,A -85,B 0,C 180,E1 -17587.468,E2 -17587.468} C_VEL
LIN {X 0,Y 277.208,Z 489.938,A -85,B 0,C 180,E1 -17591.236,E2 -17591.236} C_VEL
LIN {X 0,Y 277.215,Z 489.951,A -85,B 0,C 180,E1 -17595.222,E2 -17595.222} C_VEL
LIN {X 0,Y 277.219,Z 489.912,A -85,B 0,C 180,E1 -17599.511,E2 -17599.511} C_VEL
LIN {X 0,Y 277.261,Z 489.936,A -85,B 0,C 180,E1 -17602.529,E2 -17602.529} C_VEL
LIN {X 0,Y 277.243,Z 489.938,A -85,B 0,C 180,E1 -17606.103,E2 -17606.103} C_VEL
LIN {X 0,Y 277.257,Z 489.892,A -85,B 0,C 180,E1 -17609.538,E2 -17609.538} C_VEL
LIN {X 0,Y 277.354,Z 489.925,A -85,B 0,C 180,E1 -17612.863,E2 -17612.863} C_VEL
LIN {X 0,Y 277.292,Z 489.938,A -85,B 0,C 180,E1 -17616.076,E2 -17616.076} C_VEL
LIN {X 0,Y 277.337,Z 489.938,A -85,B 0,C 180,E1 -17620.765,E2 -17620.765} C_VEL
LIN {X 0,Y 277.422,Z 489.918,A -85,B 0,C 180,E1 -17625.325,E2 -17625.325} C_VEL
LIN {X 0,Y 277.442,Z 489.911,A -85,B 0,C 180,E1 -17629.059,E2 -17629.059} C_VEL
LIN {X 0,Y 276.825,Z 489.984,A -85,B 0,C 180,E1 -17630.272,E2 -17630.272} C_VEL
LIN {X 0,Y 273.997,Z 490.347,A -85,B 0,C 180,E1 -17632.249,E2 -17632.249} C_VEL
LIN {X 0,Y 271.561,Z 490.656,A -85,B 0,C 180,E1 -17633.855,E2 -17633.855} C_VEL
LIN {X 0,Y 270.505,Z 490.783,A -85,B 0,C 180,E1 -17635.099,E2 -17635.099} C_VEL
LIN {X 0,Y 270.416,Z 490.789,A -85,B 0,C 180,E1 -17635.521,E2 -17635.521} C_VEL
LIN {X 0,Y 270.782,Z 490.739,A -85,B 0,C 180,E1 -17638.513,E2 -17638.513} C_VEL
LIN {X 0,Y 270.782,Z 490.75,A -85,B 0,C 180,E1 -17641.487,E2 -17641.487} C_VEL
LIN {X 0,Y 270.593,Z 490.779,A -85,B 0,C 180,E1 -17647.462,E2 -17647.462} C_VEL
LIN {X 0,Y 270.407,Z 490.783,A -85,B 0,C 180,E1 -17650.482,E2 -17650.482} C_VEL
LIN {X 0,Y 270.397,Z 490.803,A -85,B 0,C 180,E1 -17655.065,E2 -17655.065} C_VEL
LIN {X 0,Y 270.294,Z 490.78,A -85,B 0,C 180,E1 -17659.756,E2 -17659.756} C_VEL
LIN {X 0,Y 270.269,Z 490.814,A -85,B 0,C 180,E1 -17664.586,E2 -17664.586} C_VEL
LIN {X 0,Y 270.267,Z 490.796,A -85,B 0,C 180,E1 -17667.909,E2 -17667.909} C_VEL
LIN {X 0,Y 270.18,Z 490.824,A -85,B 0,C 180,E1 -17671.349,E2 -17671.349} C_VEL
LIN {X 0,Y 270.197,Z 490.823,A -85,B 0,C 180,E1 -17674.906,E2 -17674.906} C_VEL
LIN {X 0,Y 270.194,Z 490.816,A -85,B 0,C 180,E1 -17678.711,E2 -17678.711} C_VEL
LIN {X 0,Y 270.174,Z 490.79,A -85,B 0,C 180,E1 -17683.252,E2 -17683.252} C_VEL
LIN {X 0,Y 270.26,Z 491.019,A -85,B 0,C 180,E1 -17687.383,E2 -17687.383} C_VEL
LIN {X 0,Y 273.397,Z 502.506,A -85,B 0,C 180,E1 -17691.116,E2 -17691.116} C_VEL
LIN {X 0,Y 276.364,Z 515.047,A -85,B 0,C 180,E1 -17694.855,E2 -17694.855} C_VEL
LIN {X 0,Y 278.373,Z 524.891,A -85,B 0,C 180,E1 -17697.616,E2 -17697.616} C_VEL
LIN {X 0,Y 277.166,Z 532.85,A -85,B 0,C 180,E1 -17699.556,E2 -17699.556} C_VEL
LIN {X 0,Y 276.664,Z 535.701,A -85,B 0,C 180,E1 -17700.202,E2 -17700.202} C_VEL
LIN {X 0,Y 280.075,Z 561.653,A -85,B 0,C 180,E1 -17701.373,E2 -17701.373} C_VEL
LIN {X 0,Y 283.505,Z 595.101,A -85,B 0,C 180,E1 -17702.666,E2 -17702.666} C_VEL
LIN {X 0,Y 284.36,Z 607.015,A -85,B 0,C 180,E1 -17703.08,E2 -17703.08} C_VEL
LIN {X 0,Y 283.074,Z 647.16,A -85,B 0,C 180,E1 -17704.099,E2 -17704.099} C_VEL
LIN {X 0,Y 282.065,Z 660.761,A -85,B 0,C 180,E1 -17704.717,E2 -17704.717} C_VEL
LIN {X 0,Y 280.618,Z 673.692,A -85,B 0,C 180,E1 -17705.592,E2 -17705.592} C_VEL
LIN {X 0,Y 278.89,Z 684.865,A -85,B 0,C 180,E1 -17706.616,E2 -17706.616} C_VEL
LIN {X 0,Y 276.829,Z 696.53,A -85,B 0,C 180,E1 -17708.009,E2 -17708.009} C_VEL
LIN {X 0,Y 274.816,Z 707.068,A -85,B 0,C 180,E1 -17709.609,E2 -17709.609} C_VEL
LIN {X 0,Y 273.179,Z 715.73,A -85,B 0,C 180,E1 -17711.242,E2 -17711.242} C_VEL
LIN {X 0,Y 271.488,Z 724.6,A -85,B 0,C 180,E1 -17713.3,E2 -17713.3} C_VEL
LIN {X 0,Y 270.335,Z 731.644,A -85,B 0,C 180,E1 -17715.317,E2 -17715.317} C_VEL
LIN {X 0,Y 269.346,Z 738.973,A -85,B 0,C 180,E1 -17717.952,E2 -17717.952} C_VEL
LIN {X 0,Y 269.024,Z 743.908,A -85,B 0,C 180,E1 -17720.224,E2 -17720.224} C_VEL
LIN {X 0,Y 269.093,Z 748.387,A -85,B 0,C 180,E1 -17722.96,E2 -17722.96} C_VEL
LIN {X 0,Y 269.47,Z 751.222,A -85,B 0,C 180,E1 -17725.513,E2 -17725.513} C_VEL
LIN {X 0,Y 269.676,Z 752.303,A -85,B 0,C 180,E1 -17727.012,E2 -17727.012} C_VEL
LIN {X 0,Y 269.982,Z 752.987,A -85,B 0,C 180,E1 -17728.508,E2 -17728.508} C_VEL
LIN {X 0,Y 270.345,Z 753.262,A -85,B 0,C 180,E1 -17730,E2 -17730} C_VEL
LIN {X 0,Y 269.984,Z 752.979,A -85,B 0,C 180,E1 -17731.492,E2 -17731.492} C_VEL
LIN {X 0,Y 269.679,Z 752.291,A -85,B 0,C 180,E1 -17732.988,E2 -17732.988} C_VEL
LIN {X 0,Y 269.478,Z 751.207,A -85,B 0,C 180,E1 -17734.487,E2 -17734.487} C_VEL
LIN {X 0,Y 269.148,Z 748.243,A -85,B 0,C 180,E1 -17737.133,E2 -17737.133} C_VEL
LIN {X 0,Y 269.025,Z 743.856,A -85,B 0,C 180,E1 -17739.776,E2 -17739.776} C_VEL
LIN {X 0,Y 269.354,Z 738.908,A -85,B 0,C 180,E1 -17742.048,E2 -17742.048} C_VEL
LIN {X 0,Y 270.338,Z 731.563,A -85,B 0,C 180,E1 -17744.683,E2 -17744.683} C_VEL
LIN {X 0,Y 271.662,Z 723.799,A -85,B 0,C 180,E1 -17746.881,E2 -17746.881} C_VEL
LIN {X 0,Y 273.154,Z 715.592,A -85,B 0,C 180,E1 -17748.76,E2 -17748.76} C_VEL
LIN {X 0,Y 275.054,Z 705.825,A -85,B 0,C 180,E1 -17750.568,E2 -17750.568} C_VEL
LIN {X 0,Y 277.079,Z 695.029,A -85,B 0,C 180,E1 -17752.166,E2 -17752.166} C_VEL
LIN {X 0,Y 278.888,Z 684.621,A -85,B 0,C 180,E1 -17753.384,E2 -17753.384} C_VEL
LIN {X 0,Y 280.76,Z 672.207,A -85,B 0,C 180,E1 -17754.493,E2 -17754.493} C_VEL
LIN {X 0,Y 282.125,Z 658.984,A -85,B 0,C 180,E1 -17755.36,E2 -17755.36} C_VEL
LIN {X 0,Y 283.077,Z 645.784,A -85,B 0,C 180,E1 -17755.923,E2 -17755.923} C_VEL
LIN {X 0,Y 284.153,Z 605.053,A -85,B 0,C 180,E1 -17756.963,E2 -17756.963} C_VEL
LIN {X 0,Y 281.434,Z 574.405,A -85,B 0,C 180,E1 -17758.09,E2 -17758.09} C_VEL
LIN {X 0,Y 277.683,Z 543.555,A -85,B 0,C 180,E1 -17759.37,E2 -17759.37} C_VEL
LIN {X 0,Y 276.668,Z 535.69,A -85,B 0,C 180,E1 -17759.766,E2 -17759.766} C_VEL
LIN {X 0,Y 278.295,Z 526.175,A -85,B 0,C 180,E1 -17762.027,E2 -17762.027} C_VEL
LIN {X 0,Y 277.862,Z 522.269,A -85,B 0,C 180,E1 -17763.071,E2 -17763.071} C_VEL
LIN {X 0,Y 275.49,Z 511.177,A -85,B 0,C 180,E1 -17766.225,E2 -17766.225} C_VEL
LIN {X 0,Y 272.595,Z 499.42,A -85,B 0,C 180,E1 -17769.806,E2 -17769.806} C_VEL
LIN {X 0,Y 270.252,Z 490.89,A -85,B 0,C 180,E1 -17772.629,E2 -17772.629} C_VEL
LIN {X 0,Y 270.174,Z 490.79,A -85,B 0,C 180,E1 -17776.748,E2 -17776.748} C_VEL
LIN {X 0,Y 270.204,Z 490.813,A -85,B 0,C 180,E1 -17781.373,E2 -17781.373} C_VEL
LIN {X 0,Y 270.197,Z 490.822,A -85,B 0,C 180,E1 -17785.094,E2 -17785.094} C_VEL
LIN {X 0,Y 270.196,Z 490.829,A -85,B 0,C 180,E1 -17789.13,E2 -17789.13} C_VEL
LIN {X 0,Y 270.26,Z 490.796,A -85,B 0,C 180,E1 -17792.145,E2 -17792.145} C_VEL
LIN {X 0,Y 270.272,Z 490.814,A -85,B 0,C 180,E1 -17795.519,E2 -17795.519} C_VEL
LIN {X 0,Y 270.294,Z 490.78,A -85,B 0,C 180,E1 -17800.244,E2 -17800.244} C_VEL
LIN {X 0,Y 270.397,Z 490.804,A -85,B 0,C 180,E1 -17804.935,E2 -17804.935} C_VEL
LIN {X 0,Y 270.407,Z 490.785,A -85,B 0,C 180,E1 -17809.518,E2 -17809.518} C_VEL
LIN {X 0,Y 270.593,Z 490.78,A -85,B 0,C 180,E1 -17812.538,E2 -17812.538} C_VEL
LIN {X 0,Y 270.782,Z 490.754,A -85,B 0,C 180,E1 -17818.513,E2 -17818.513} C_VEL
LIN {X 0,Y 270.782,Z 490.742,A -85,B 0,C 180,E1 -17821.487,E2 -17821.487} C_VEL
LIN {X 0,Y 270.594,Z 490.772,A -85,B 0,C 180,E1 -17827.462,E2 -17827.462} C_VEL
LIN {X 0,Y 270.407,Z 490.784,A -85,B 0,C 180,E1 -17830.483,E2 -17830.483} C_VEL
LIN {X 0,Y 270.391,Z 490.789,A -85,B 0,C 180,E1 -17835.065,E2 -17835.065} C_VEL
LIN {X 0,Y 270.295,Z 490.815,A -85,B 0,C 180,E1 -17839.756,E2 -17839.756} C_VEL
LIN {X 0,Y 270.233,Z 490.821,A -85,B 0,C 180,E1 -17844.59,E2 -17844.59} C_VEL
LIN {X 0,Y 270.266,Z 490.796,A -85,B 0,C 180,E1 -17847.909,E2 -17847.909} C_VEL
LIN {X 0,Y 270.18,Z 490.774,A -85,B 0,C 180,E1 -17851.349,E2 -17851.349} C_VEL
LIN {X 0,Y 270.198,Z 490.825,A -85,B 0,C 180,E1 -17854.906,E2 -17854.906} C_VEL
LIN {X 0,Y 270.194,Z 490.793,A -85,B 0,C 180,E1 -17858.711,E2 -17858.711} C_VEL
LIN {X 0,Y 270.169,Z 490.828,A -85,B 0,C 180,E1 -17863.251,E2 -17863.251} C_VEL
LIN {X 0,Y 270.172,Z 490.801,A -85,B 0,C 180,E1 -17867.443,E2 -17867.443} C_VEL
LIN {X 0,Y 270.206,Z 490.821,A -85,B 0,C 180,E1 -17871.375,E2 -17871.375} C_VEL
LIN {X 0,Y 270.201,Z 490.746,A -85,B 0,C 180,E1 -17875.095,E2 -17875.095} C_VEL
LIN {X 0,Y 270.2,Z 490.815,A -85,B 0,C 180,E1 -17879.131,E2 -17879.131} C_VEL
LIN {X 0,Y 270.278,Z 491.086,A -85,B 0,C 180,E1 -17880.045,E2 -17880.045} C_VEL
LIN {X 0,Y 270.621,Z 492.28,A -85,B 0,C 180,E1 -17880.293,E2 -17880.293} C_VEL
LIN {X 0,Y 279.377,Z 508.8,A -85,B 0,C 180,E1 -17881.844,E2 -17881.844} C_VEL
LIN {X 0,Y 286.401,Z 524.263,A -85,B 0,C 180,E1 -17883.056,E2 -17883.056} C_VEL
LIN {X 0,Y 285.571,Z 569.435,A -85,B 0,C 180,E1 -17884.223,E2 -17884.223} C_VEL
LIN {X 0,Y 285.261,Z 583.166,A -85,B 0,C 180,E1 -17884.772,E2 -17884.772} C_VEL
LIN {X 0,Y 284.485,Z 595.923,A -85,B 0,C 180,E1 -17885.557,E2 -17885.557} C_VEL
LIN {X 0,Y 283.389,Z 608.163,A -85,B 0,C 180,E1 -17886.623,E2 -17886.623} C_VEL
LIN {X 0,Y 282.129,Z 618.428,A -85,B 0,C 180,E1 -17887.77,E2 -17887.77} C_VEL
LIN {X 0,Y 280.488,Z 629.168,A -85,B 0,C 180,E1 -17889.273,E2 -17889.273} C_VEL
LIN {X 0,Y 278.923,Z 638.361,A -85,B 0,C 180,E1 -17890.88,E2 -17890.88} C_VEL
LIN {X 0,Y 277.428,Z 646.714,A -85,B 0,C 180,E1 -17892.683,E2 -17892.683} C_VEL
LIN {X 0,Y 275.752,Z 654.826,A -85,B 0,C 180,E1 -17894.857,E2 -17894.857} C_VEL
LIN {X 0,Y 274.154,Z 661.933,A -85,B 0,C 180,E1 -17897.26,E2 -17897.26} C_VEL
LIN {X 0,Y 273.05,Z 667.304,A -85,B 0,C 180,E1 -17899.62,E2 -17899.62} C_VEL
LIN {X 0,Y 271.994,Z 671.194,A -85,B 0,C 180,E1 -17901.83,E2 -17901.83} C_VEL
LIN {X 0,Y 271.213,Z 674.062,A -85,B 0,C 180,E1 -17904.051,E2 -17904.051} C_VEL
LIN {X 0,Y 271.05,Z 675.405,A -85,B 0,C 180,E1 -17905.539,E2 -17905.539} C_VEL
LIN {X 0,Y 270.93,Z 676.359,A -85,B 0,C 180,E1 -17907.026,E2 -17907.026} C_VEL
LIN {X 0,Y 270.719,Z 677.186,A -85,B 0,C 180,E1 -17910,E2 -17910} C_VEL
LIN {X 0,Y 270.923,Z 676.421,A -85,B 0,C 180,E1 -17912.974,E2 -17912.974} C_VEL
LIN {X 0,Y 271.199,Z 674.187,A -85,B 0,C 180,E1 -17915.95,E2 -17915.95} C_VEL
LIN {X 0,Y 271.987,Z 671.364,A -85,B 0,C 180,E1 -17918.17,E2 -17918.17} C_VEL
LIN {X 0,Y 273.025,Z 667.534,A -85,B 0,C 180,E1 -17920.38,E2 -17920.38} C_VEL
LIN {X 0,Y 274.072,Z 662.453,A -85,B 0,C 180,E1 -17922.664,E2 -17922.664} C_VEL
LIN {X 0,Y 275.445,Z 656.419,A -85,B 0,C 180,E1 -17924.782,E2 -17924.782} C_VEL
LIN {X 0,Y 277.117,Z 648.634,A -85,B 0,C 180,E1 -17926.956,E2 -17926.956} C_VEL
LIN {X 0,Y 278.879,Z 638.959,A -85,B 0,C 180,E1 -17929.123,E2 -17929.123} C_VEL
LIN {X 0,Y 280.445,Z 629.909,A -85,B 0,C 180,E1 -17930.73,E2 -17930.73} C_VEL
LIN {X 0,Y 282.104,Z 619.393,A -85,B 0,C 180,E1 -17932.222,E2 -17932.222} C_VEL
LIN {X 0,Y 283.507,Z 607.866,A -85,B 0,C 180,E1 -17933.524,E2 -17933.524} C_VEL
LIN {X 0,Y 284.697,Z 596.571,A -85,B 0,C 180,E1 -17934.491,E2 -17934.491} C_VEL
LIN {X 0,Y 285.26,Z 583.903,A -85,B 0,C 180,E1 -17935.313,E2 -17935.313} C_VEL
LIN {X 0,Y 285.585,Z 570.117,A -85,B 0,C 180,E1 -17935.877,E2 -17935.877} C_VEL
LIN {X 0,Y 286.33,Z 530.623,A -85,B 0,C 180,E1 -17936.9,E2 -17936.9} C_VEL
LIN {X 0,Y 286.459,Z 524.273,A -85,B 0,C 180,E1 -17937.062,E2 -17937.062} C_VEL
LIN {X 0,Y 278.862,Z 507.802,A -85,B 0,C 180,E1 -17938.372,E2 -17938.372} C_VEL
LIN {X 0,Y 271.147,Z 493.404,A -85,B 0,C 180,E1 -17939.726,E2 -17939.726} C_VEL
LIN {X 0,Y 270.364,Z 491.4,A -85,B 0,C 180,E1 -17939.979,E2 -17939.979} C_VEL
LIN {X 0,Y 270.237,Z 490.882,A -85,B 0,C 180,E1 -17940.257,E2 -17940.257} C_VEL
LIN {X 0,Y 270.215,Z 490.818,A -85,B 0,C 180,E1 -17943.665,E2 -17943.665} C_VEL
LIN {X 0,Y 270.216,Z 490.805,A -85,B 0,C 180,E1 -17946.74,E2 -17946.74} C_VEL
LIN {X 0,Y 270.167,Z 490.817,A -85,B 0,C 180,E1 -17951.027,E2 -17951.027} C_VEL
LIN {X 0,Y 270.164,Z 490.831,A -85,B 0,C 180,E1 -17955.382,E2 -17955.382} C_VEL
LIN {X 0,Y 270.17,Z 490.789,A -85,B 0,C 180,E1 -17959.433,E2 -17959.433} C_VEL
LIN {X 0,Y 270.221,Z 490.826,A -85,B 0,C 180,E1 -17963.73,E2 -17963.73} C_VEL
LIN {X 0,Y 270.199,Z 490.8,A -85,B 0,C 180,E1 -17966.892,E2 -17966.892} C_VEL
LIN {X 0,Y 270.192,Z 490.776,A -85,B 0,C 180,E1 -17970.382,E2 -17970.382} C_VEL
LIN {X 0,Y 270.257,Z 490.819,A -85,B 0,C 180,E1 -17973.763,E2 -17973.763} C_VEL
LIN {X 0,Y 270.205,Z 490.812,A -85,B 0,C 180,E1 -17977.036,E2 -17977.036} C_VEL
LIN {X 0,Y 270.295,Z 490.815,A -85,B 0,C 180,E1 -17980.244,E2 -17980.244} C_VEL
LIN {X 0,Y 270.391,Z 490.79,A -85,B 0,C 180,E1 -17984.935,E2 -17984.935} C_VEL
LIN {X 0,Y 270.436,Z 490.781,A -85,B 0,C 180,E1 -17989.519,E2 -17989.519} C_VEL
LIN {X 0,Y 270.605,Z 490.77,A -85,B 0,C 180,E1 -17992.539,E2 -17992.539} C_VEL
LIN {X 0,Y 270.416,Z 490.789,A -85,B 0,C 180,E1 -17995.521,E2 -17995.521} C_VEL
LIN {X 0,Y 269.791,Z 490.871,A -85,B 0,C 180,E1 -17996.768,E2 -17996.768} C_VEL
LIN {X 0,Y 267.137,Z 491.208,A -85,B 0,C 180,E1 -17998.807,E2 -17998.807} C_VEL
LIN {X 0,Y 264.025,Z 491.594,A -85,B 0,C 180,E1 -18001.309,E2 -18001.309} C_VEL
LIN {X 0,Y 263.644,Z 491.631,A -85,B 0,C 180,E1 -18002.172,E2 -18002.172} C_VEL
LIN {X 0,Y 263.553,Z 491.656,A -85,B 0,C 180,E1 -18007.662,E2 -18007.662} C_VEL
LIN {X 0,Y 263.349,Z 491.661,A -85,B 0,C 180,E1 -18010.767,E2 -18010.767} C_VEL
LIN {X 0,Y 263.345,Z 491.677,A -85,B 0,C 180,E1 -18015.478,E2 -18015.478} C_VEL
LIN {X 0,Y 263.257,Z 491.662,A -85,B 0,C 180,E1 -18020.307,E2 -18020.307} C_VEL
LIN {X 0,Y 263.204,Z 491.681,A -85,B 0,C 180,E1 -18025.292,E2 -18025.292} C_VEL
LIN {X 0,Y 263.175,Z 491.691,A -85,B 0,C 180,E1 -18028.73,E2 -18028.73} C_VEL
LIN {X 0,Y 263.129,Z 491.692,A -85,B 0,C 180,E1 -18032.289,E2 -18032.289} C_VEL
LIN {X 0,Y 263.186,Z 491.697,A -85,B 0,C 180,E1 -18036.766,E2 -18036.766} C_VEL
LIN {X 0,Y 263.122,Z 491.693,A -85,B 0,C 180,E1 -18041.595,E2 -18041.595} C_VEL
LIN {X 0,Y 263.142,Z 491.683,A -85,B 0,C 180,E1 -18046.021,E2 -18046.021} C_VEL
LIN {X 0,Y 263.201,Z 491.978,A -85,B 0,C 180,E1 -18046.619,E2 -18046.619} C_VEL
LIN {X 0,Y 266,Z 501.972,A -85,B 0,C 180,E1 -18050.015,E2 -18050.015} C_VEL
LIN {X 0,Y 268.865,Z 513.703,A -85,B 0,C 180,E1 -18053.679,E2 -18053.679} C_VEL
LIN {X 0,Y 271.241,Z 525.18,A -85,B 0,C 180,E1 -18057.036,E2 -18057.036} C_VEL
LIN {X 0,Y 271.494,Z 526.881,A -85,B 0,C 180,E1 -18057.512,E2 -18057.512} C_VEL
LIN {X 0,Y 270.158,Z 534.7,A -85,B 0,C 180,E1 -18059.414,E2 -18059.414} C_VEL
LIN {X 0,Y 273.81,Z 562.4,A -85,B 0,C 180,E1 -18060.706,E2 -18060.706} C_VEL
LIN {X 0,Y 277.457,Z 599.112,A -85,B 0,C 180,E1 -18062.159,E2 -18062.159} C_VEL
LIN {X 0,Y 277.914,Z 609.524,A -85,B 0,C 180,E1 -18062.502,E2 -18062.502} C_VEL
LIN {X 0,Y 276.653,Z 646.99,A -85,B 0,C 180,E1 -18063.488,E2 -18063.488} C_VEL
LIN {X 0,Y 275.582,Z 660.569,A -85,B 0,C 180,E1 -18064.131,E2 -18064.131} C_VEL
LIN {X 0,Y 274.201,Z 672.705,A -85,B 0,C 180,E1 -18064.982,E2 -18064.982} C_VEL
LIN {X 0,Y 272.355,Z 683.867,A -85,B 0,C 180,E1 -18066.02,E2 -18066.02} C_VEL
LIN {X 0,Y 270.211,Z 695.528,A -85,B 0,C 180,E1 -18067.441,E2 -18067.441} C_VEL
LIN {X 0,Y 268.169,Z 706.073,A -85,B 0,C 180,E1 -18069.08,E2 -18069.08} C_VEL
LIN {X 0,Y 266.417,Z 714.727,A -85,B 0,C 180,E1 -18070.747,E2 -18070.747} C_VEL
LIN {X 0,Y 264.889,Z 722.76,A -85,B 0,C 180,E1 -18072.634,E2 -18072.634} C_VEL
LIN {X 0,Y 263.752,Z 727.929,A -85,B 0,C 180,E1 -18074.079,E2 -18074.079} C_VEL
LIN {X 0,Y 262.712,Z 735.044,A -85,B 0,C 180,E1 -18076.463,E2 -18076.463} C_VEL
LIN {X 0,Y 262.036,Z 741.397,A -85,B 0,C 180,E1 -18079.179,E2 -18079.179} C_VEL
LIN {X 0,Y 261.951,Z 745.582,A -85,B 0,C 180,E1 -18081.515,E2 -18081.515} C_VEL
LIN {X 0,Y 262.11,Z 748.707,A -85,B 0,C 180,E1 -18083.843,E2 -18083.843} C_VEL
LIN {X 0,Y 262.392,Z 750.224,A -85,B 0,C 180,E1 -18085.391,E2 -18085.391} C_VEL
LIN {X 0,Y 262.615,Z 751.309,A -85,B 0,C 180,E1 -18086.932,E2 -18086.932} C_VEL
LIN {X 0,Y 262.923,Z 751.994,A -85,B 0,C 180,E1 -18088.468,E2 -18088.468} C_VEL
LIN {X 0,Y 263.309,Z 752.273,A -85,B 0,C 180,E1 -18090,E2 -18090} C_VEL
LIN {X 0,Y 262.925,Z 751.986,A -85,B 0,C 180,E1 -18091.532,E2 -18091.532} C_VEL
LIN {X 0,Y 262.618,Z 751.297,A -85,B 0,C 180,E1 -18093.068,E2 -18093.068} C_VEL
LIN {X 0,Y 262.403,Z 750.208,A -85,B 0,C 180,E1 -18094.609,E2 -18094.609} C_VEL
LIN {X 0,Y 262.073,Z 747.465,A -85,B 0,C 180,E1 -18097.147,E2 -18097.147} C_VEL
LIN {X 0,Y 261.946,Z 744.24,A -85,B 0,C 180,E1 -18099.264,E2 -18099.264} C_VEL
LIN {X 0,Y 262.182,Z 739.674,A -85,B 0,C 180,E1 -18101.598,E2 -18101.598} C_VEL
LIN {X 0,Y 262.881,Z 733.925,A -85,B 0,C 180,E1 -18103.922,E2 -18103.922} C_VEL
LIN {X 0,Y 263.855,Z 727.627,A -85,B 0,C 180,E1 -18105.983,E2 -18105.983} C_VEL
LIN {X 0,Y 265.452,Z 719.6,A -85,B 0,C 180,E1 -18108.124,E2 -18108.124} C_VEL
LIN {X 0,Y 267.152,Z 710.938,A -85,B 0,C 180,E1 -18109.998,E2 -18109.998} C_VEL
LIN {X 0,Y 269.314,Z 700.303,A -85,B 0,C 180,E1 -18111.83,E2 -18111.83} C_VEL
LIN {X 0,Y 271.313,Z 689.816,A -85,B 0,C 180,E1 -18113.267,E2 -18113.267} C_VEL
LIN {X 0,Y 273.285,Z 678.344,A -85,B 0,C 180,E1 -18114.499,E2 -18114.499} C_VEL
LIN {X 0,Y 274.888,Z 666.54,A -85,B 0,C 180,E1 -18115.457,E2 -18115.457} C_VEL
LIN {X 0,Y 276.116,Z 653.802,A -85,B 0,C 180,E1 -18116.199,E2 -18116.199} C_VEL
LIN {X 0,Y 276.831,Z 640.73,A -85,B 0,C 180,E1 -18116.688,E2 -18116.688} C_VEL
LIN {X 0,Y 277.755,Z 605.816,A -85,B 0,C 180,E1 -18117.585,E2 -18117.585} C_VEL
LIN {X 0,Y 275.405,Z 578.081,A -85,B 0,C 180,E1 -18118.627,E2 -18118.627} C_VEL
LIN {X 0,Y 271.955,Z 548.234,A -85,B 0,C 180,E1 -18119.886,E2 -18119.886} C_VEL
LIN {X 0,Y 270.093,Z 534.75,A -85,B 0,C 180,E1 -18120.548,E2 -18120.548} C_VEL
LIN {X 0,Y 271.461,Z 526.747,A -85,B 0,C 180,E1 -18122.493,E2 -18122.493} C_VEL
LIN {X 0,Y 269.842,Z 518.148,A -85,B 0,C 180,E1 -18124.958,E2 -18124.958} C_VEL
LIN {X 0,Y 267.219,Z 506.722,A -85,B 0,C 180,E1 -18128.415,E2 -18128.415} C_VEL
LIN {X 0,Y 264.401,Z 496.058,A -85,B 0,C 180,E1 -18131.904,E2 -18131.904} C_VEL
LIN {X 0,Y 263.178,Z 491.747,A -85,B 0,C 180,E1 -18133.446,E2 -18133.446} C_VEL
LIN {X 0,Y 263.131,Z 491.664,A -85,B 0,C 180,E1 -18136.148,E2 -18136.148} C_VEL
LIN {X 0,Y 263.103,Z 491.709,A -85,B 0,C 180,E1 -18140.127,E2 -18140.127} C_VEL
LIN {X 0,Y 263.159,Z 491.706,A -85,B 0,C 180,E1 -18144.017,E2 -18144.017} C_VEL
LIN {X 0,Y 263.129,Z 491.693,A -85,B 0,C 180,E1 -18147.711,E2 -18147.711} C_VEL
LIN {X 0,Y 263.197,Z 491.679,A -85,B 0,C 180,E1 -18151.783,E2 -18151.783} C_VEL
LIN {X 0,Y 263.221,Z 491.687,A -85,B 0,C 180,E1 -18155.2,E2 -18155.2} C_VEL
LIN {X 0,Y 263.257,Z 491.661,A -85,B 0,C 180,E1 -18159.693,E2 -18159.693} C_VEL
LIN {X 0,Y 263.345,Z 491.677,A -85,B 0,C 180,E1 -18164.522,E2 -18164.522} C_VEL
LIN {X 0,Y 263.349,Z 491.662,A -85,B 0,C 180,E1 -18169.233,E2 -18169.233} C_VEL
LIN {X 0,Y 263.553,Z 491.657,A -85,B 0,C 180,E1 -18172.338,E2 -18172.338} C_VEL
LIN {X 0,Y 263.746,Z 491.63,A -85,B 0,C 180,E1 -18178.473,E2 -18178.473} C_VEL
LIN {X 0,Y 263.746,Z 491.617,A -85,B 0,C 180,E1 -18181.527,E2 -18181.527} C_VEL
LIN {X 0,Y 263.553,Z 491.649,A -85,B 0,C 180,E1 -18187.662,E2 -18187.662} C_VEL
LIN {X 0,Y 263.349,Z 491.666,A -85,B 0,C 180,E1 -18190.767,E2 -18190.767} C_VEL
LIN {X 0,Y 263.339,Z 491.665,A -85,B 0,C 180,E1 -18195.479,E2 -18195.479} C_VEL
LIN {X 0,Y 263.257,Z 491.691,A -85,B 0,C 180,E1 -18200.307,E2 -18200.307} C_VEL
LIN {X 0,Y 263.188,Z 491.701,A -85,B 0,C 180,E1 -18205.294,E2 -18205.294} C_VEL
LIN {X 0,Y 263.162,Z 491.665,A -85,B 0,C 180,E1 -18208.732,E2 -18208.732} C_VEL
LIN {X 0,Y 263.129,Z 491.661,A -85,B 0,C 180,E1 -18212.289,E2 -18212.289} C_VEL
LIN {X 0,Y 263.178,Z 491.697,A -85,B 0,C 180,E1 -18216.764,E2 -18216.764} C_VEL
LIN {X 0,Y 263.122,Z 491.676,A -85,B 0,C 180,E1 -18221.594,E2 -18221.594} C_VEL
LIN {X 0,Y 263.126,Z 491.709,A -85,B 0,C 180,E1 -18223.984,E2 -18223.984} C_VEL
LIN {X 0,Y 263.123,Z 491.683,A -85,B 0,C 180,E1 -18228.407,E2 -18228.407} C_VEL
LIN {X 0,Y 263.159,Z 491.677,A -85,B 0,C 180,E1 -18232.104,E2 -18232.104} C_VEL
LIN {X 0,Y 263.15,Z 491.623,A -85,B 0,C 180,E1 -18235.886,E2 -18235.886} C_VEL
LIN {X 0,Y 263.181,Z 491.849,A -85,B 0,C 180,E1 -18239.067,E2 -18239.067} C_VEL
LIN {X 0,Y 263.429,Z 492.87,A -85,B 0,C 180,E1 -18239.366,E2 -18239.366} C_VEL
LIN {X 0,Y 272.983,Z 510.671,A -85,B 0,C 180,E1 -18241.148,E2 -18241.148} C_VEL
LIN {X 0,Y 280.11,Z 526.092,A -85,B 0,C 180,E1 -18242.423,E2 -18242.423} C_VEL
LIN {X 0,Y 279.268,Z 567.636,A -85,B 0,C 180,E1 -18243.515,E2 -18243.515} C_VEL
LIN {X 0,Y 279.01,Z 581.116,A -85,B 0,C 180,E1 -18243.997,E2 -18243.997} C_VEL
LIN {X 0,Y 278.297,Z 594.353,A -85,B 0,C 180,E1 -18244.777,E2 -18244.777} C_VEL
LIN {X 0,Y 277.227,Z 606.917,A -85,B 0,C 180,E1 -18245.823,E2 -18245.823} C_VEL
LIN {X 0,Y 275.831,Z 618.357,A -85,B 0,C 180,E1 -18247.085,E2 -18247.085} C_VEL
LIN {X 0,Y 274.338,Z 627.849,A -85,B 0,C 180,E1 -18248.392,E2 -18248.392} C_VEL
LIN {X 0,Y 272.64,Z 637.439,A -85,B 0,C 180,E1 -18250.029,E2 -18250.029} C_VEL
LIN {X 0,Y 270.987,Z 646.14,A -85,B 0,C 180,E1 -18251.868,E2 -18251.868} C_VEL
LIN {X 0,Y 269.262,Z 654.609,A -85,B 0,C 180,E1 -18254.094,E2 -18254.094} C_VEL
LIN {X 0,Y 267.658,Z 661.365,A -85,B 0,C 180,E1 -18256.331,E2 -18256.331} C_VEL
LIN {X 0,Y 266.498,Z 666.739,A -85,B 0,C 180,E1 -18258.593,E2 -18258.593} C_VEL
LIN {X 0,Y 265.285,Z 670.992,A -85,B 0,C 180,E1 -18260.854,E2 -18260.854} C_VEL
LIN {X 0,Y 264.707,Z 673.229,A -85,B 0,C 180,E1 -18262.372,E2 -18262.372} C_VEL
LIN {X 0,Y 264.222,Z 675.051,A -85,B 0,C 180,E1 -18263.893,E2 -18263.893} C_VEL
LIN {X 0,Y 264.042,Z 676.393,A -85,B 0,C 180,E1 -18265.42,E2 -18265.42} C_VEL
LIN {X 0,Y 263.918,Z 677.347,A -85,B 0,C 180,E1 -18266.947,E2 -18266.947} C_VEL
LIN {X 0,Y 263.692,Z 678.174,A -85,B 0,C 180,E1 -18270,E2 -18270} C_VEL
LIN {X 0,Y 263.911,Z 677.408,A -85,B 0,C 180,E1 -18273.053,E2 -18273.053} C_VEL
LIN {X 0,Y 264.207,Z 675.175,A -85,B 0,C 180,E1 -18276.108,E2 -18276.108} C_VEL
LIN {X 0,Y 265.032,Z 672.351,A -85,B 0,C 180,E1 -18278.386,E2 -18278.386} C_VEL
LIN {X 0,Y 266.115,Z 668.521,A -85,B 0,C 180,E1 -18280.653,E2 -18280.653} C_VEL
LIN {X 0,Y 267.219,Z 663.439,A -85,B 0,C 180,E1 -18282.994,E2 -18282.994} C_VEL
LIN {X 0,Y 268.656,Z 657.405,A -85,B 0,C 180,E1 -18285.165,E2 -18285.165} C_VEL
LIN {X 0,Y 270.402,Z 649.62,A -85,B 0,C 180,E1 -18287.391,E2 -18287.391} C_VEL
LIN {X 0,Y 272.247,Z 639.944,A -85,B 0,C 180,E1 -18289.608,E2 -18289.608} C_VEL
LIN {X 0,Y 273.884,Z 630.893,A -85,B 0,C 180,E1 -18291.25,E2 -18291.25} C_VEL
LIN {X 0,Y 275.611,Z 620.376,A -85,B 0,C 180,E1 -18292.775,E2 -18292.775} C_VEL
LIN {X 0,Y 277.106,Z 608.691,A -85,B 0,C 180,E1 -18294.119,E2 -18294.119} C_VEL
LIN {X 0,Y 278.355,Z 597.209,A -85,B 0,C 180,E1 -18295.117,E2 -18295.117} C_VEL
LIN {X 0,Y 278.895,Z 585.133,A -85,B 0,C 180,E1 -18295.919,E2 -18295.919} C_VEL
LIN {X 0,Y 279.22,Z 571.952,A -85,B 0,C 180,E1 -18296.483,E2 -18296.483} C_VEL
LIN {X 0,Y 280.1,Z 529.84,A -85,B 0,C 180,E1 -18297.598,E2 -18297.598} C_VEL
LIN {X 0,Y 280.167,Z 526.135,A -85,B 0,C 180,E1 -18297.696,E2 -18297.696} C_VEL
LIN {X 0,Y 272.603,Z 509.907,A -85,B 0,C 180,E1 -18299.051,E2 -18299.051} C_VEL
LIN {X 0,Y 264.498,Z 495.042,A -85,B 0,C 180,E1 -18300.533,E2 -18300.533} C_VEL
LIN {X 0,Y 263.318,Z 492.55,A -85,B 0,C 180,E1 -18300.82,E2 -18300.82} C_VEL
LIN {X 0,Y 263.157,Z 491.76,A -85,B 0,C 180,E1 -18301.161,E2 -18301.161} C_VEL
LIN {X 0,Y 263.173,Z 491.701,A -85,B 0,C 180,E1 -18304.121,E2 -18304.121} C_VEL
LIN {X 0,Y 263.158,Z 491.688,A -85,B 0,C 180,E1 -18307.896,E2 -18307.896} C_VEL
LIN {X 0,Y 263.123,Z 491.683,A -85,B 0,C 180,E1 -18311.892,E2 -18311.892} C_VEL
LIN {X 0,Y 263.127,Z 491.711,A -85,B 0,C 180,E1 -18316.149,E2 -18316.149} C_VEL
LIN {X 0,Y 263.102,Z 491.667,A -85,B 0,C 180,E1 -18320.127,E2 -18320.127} C_VEL
LIN {X 0,Y 263.159,Z 491.705,A -85,B 0,C 180,E1 -18324.017,E2 -18324.017} C_VEL
LIN {X 0,Y 263.129,Z 491.662,A -85,B 0,C 180,E1 -18327.711,E2 -18327.711} C_VEL
LIN {X 0,Y 263.192,Z 491.669,A -85,B 0,C 180,E1 -18331.784,E2 -18331.784} C_VEL
LIN {X 0,Y 263.196,Z 491.7,A -85,B 0,C 180,E1 -18335.212,E2 -18335.212} C_VEL
LIN {X 0,Y 263.257,Z 491.69,A -85,B 0,C 180,E1 -18339.693,E2 -18339.693} C_VEL
LIN {X 0,Y 263.339,Z 491.665,A -85,B 0,C 180,E1 -18344.521,E2 -18344.521} C_VEL
LIN {X 0,Y 263.368,Z 491.664,A -85,B 0,C 180,E1 -18349.234,E2 -18349.234} C_VEL
LIN {X 0,Y 263.567,Z 491.646,A -85,B 0,C 180,E1 -18352.338,E2 -18352.338} C_VEL
LIN {X 0,Y 263.746,Z 491.614,A -85,B 0,C 180,E1 -18358.473,E2 -18358.473} C_VEL
LIN {X 0,Y 263.746,Z 491.626,A -85,B 0,C 180,E1 -18361.527,E2 -18361.527} C_VEL
LIN {X 0,Y 263.644,Z 491.631,A -85,B 0,C 180,E1 -18362.172,E2 -18362.172} C_VEL
LIN {X 0,Y 262.863,Z 491.722,A -85,B 0,C 180,E1 -18363.446,E2 -18363.446} C_VEL
LIN {X 0,Y 259.961,Z 492.087,A -85,B 0,C 180,E1 -18365.522,E2 -18365.522} C_VEL
LIN {X 0,Y 257.559,Z 492.4,A -85,B 0,C 180,E1 -18367.211,E2 -18367.211} C_VEL
LIN {X 0,Y 256.524,Z 492.528,A -85,B 0,C 180,E1 -18368.52,E2 -18368.52} C_VEL
LIN {X 0,Y 256.434,Z 492.532,A -85,B 0,C 180,E1 -18368.964,E2 -18368.964} C_VEL
LIN {X 0,Y 256.289,Z 492.554,A -85,B 0,C 180,E1 -18372.672,E2 -18372.672} C_VEL
LIN {X 0,Y 256.277,Z 492.55,A -85,B 0,C 180,E1 -18376.302,E2 -18376.302} C_VEL
LIN {X 0,Y 256.15,Z 492.561,A -85,B 0,C 180,E1 -18381.119,E2 -18381.119} C_VEL
LIN {X 0,Y 256.184,Z 492.557,A -85,B 0,C 180,E1 -18385.139,E2 -18385.139} C_VEL
LIN {X 0,Y 256.11,Z 492.581,A -85,B 0,C 180,E1 -18389.6,E2 -18389.6} C_VEL
LIN {X 0,Y 256.064,Z 492.567,A -85,B 0,C 180,E1 -18393.293,E2 -18393.293} C_VEL
LIN {X 0,Y 256.116,Z 492.571,A -85,B 0,C 180,E1 -18397.273,E2 -18397.273} C_VEL
LIN {X 0,Y 256.053,Z 492.582,A -85,B 0,C 180,E1 -18401.204,E2 -18401.204} C_VEL
LIN {X 0,Y 256.072,Z 492.605,A -85,B 0,C 180,E1 -18405.527,E2 -18405.527} C_VEL
LIN {X 0,Y 256.267,Z 493.44,A -85,B 0,C 180,E1 -18406.006,E2 -18406.006} C_VEL
LIN {X 0,Y 258.681,Z 501.732,A -85,B 0,C 180,E1 -18408.936,E2 -18408.936} C_VEL
LIN {X 0,Y 261.005,Z 510.898,A -85,B 0,C 180,E1 -18411.961,E2 -18411.961} C_VEL
LIN {X 0,Y 263.147,Z 520.553,A -85,B 0,C 180,E1 -18414.958,E2 -18414.958} C_VEL
LIN {X 0,Y 264.481,Z 527.408,A -85,B 0,C 180,E1 -18416.994,E2 -18416.994} C_VEL
LIN {X 0,Y 264.265,Z 530.675,A -85,B 0,C 180,E1 -18417.868,E2 -18417.868} C_VEL
LIN {X 0,Y 263.706,Z 533.798,A -85,B 0,C 180,E1 -18418.599,E2 -18418.599} C_VEL
LIN {X 0,Y 267.664,Z 564.306,A -85,B 0,C 180,E1 -18420.052,E2 -18420.052} C_VEL
LIN {X 0,Y 271.01,Z 598.511,A -85,B 0,C 180,E1 -18421.449,E2 -18421.449} C_VEL
LIN {X 0,Y 271.605,Z 609.357,A -85,B 0,C 180,E1 -18421.831,E2 -18421.831} C_VEL
LIN {X 0,Y 270.311,Z 645.8,A -85,B 0,C 180,E1 -18422.806,E2 -18422.806} C_VEL
LIN {X 0,Y 269.16,Z 659.67,A -85,B 0,C 180,E1 -18423.473,E2 -18423.473} C_VEL
LIN {X 0,Y 267.795,Z 671.715,A -85,B 0,C 180,E1 -18424.341,E2 -18424.341} C_VEL
LIN {X 0,Y 265.884,Z 682.873,A -85,B 0,C 180,E1 -18425.399,E2 -18425.399} C_VEL
LIN {X 0,Y 263.636,Z 694.529,A -85,B 0,C 180,E1 -18426.847,E2 -18426.847} C_VEL
LIN {X 0,Y 261.502,Z 705.071,A -85,B 0,C 180,E1 -18428.52,E2 -18428.52} C_VEL
LIN {X 0,Y 259.68,Z 713.725,A -85,B 0,C 180,E1 -18430.227,E2 -18430.227} C_VEL
LIN {X 0,Y 258.077,Z 721.757,A -85,B 0,C 180,E1 -18432.16,E2 -18432.16} C_VEL
LIN {X 0,Y 256.763,Z 727.269,A -85,B 0,C 180,E1 -18433.746,E2 -18433.746} C_VEL
LIN {X 0,Y 255.753,Z 734.039,A -85,B 0,C 180,E1 -18436.087,E2 -18436.087} C_VEL
LIN {X 0,Y 255,Z 740.391,A -85,B 0,C 180,E1 -18438.877,E2 -18438.877} C_VEL
LIN {X 0,Y 254.867,Z 744.575,A -85,B 0,C 180,E1 -18441.277,E2 -18441.277} C_VEL
LIN {X 0,Y 255.042,Z 747.707,A -85,B 0,C 180,E1 -18443.672,E2 -18443.672} C_VEL
LIN {X 0,Y 255.318,Z 749.226,A -85,B 0,C 180,E1 -18445.263,E2 -18445.263} C_VEL
LIN {X 0,Y 255.554,Z 750.315,A -85,B 0,C 180,E1 -18446.847,E2 -18446.847} C_VEL
LIN {X 0,Y 255.863,Z 751.001,A -85,B 0,C 180,E1 -18448.426,E2 -18448.426} C_VEL
LIN {X 0,Y 256.271,Z 751.283,A -85,B 0,C 180,E1 -18450,E2 -18450} C_VEL
LIN {X 0,Y 255.865,Z 750.993,A -85,B 0,C 180,E1 -18451.574,E2 -18451.574} C_VEL
LIN {X 0,Y 255.558,Z 750.302,A -85,B 0,C 180,E1 -18453.153,E2 -18453.153} C_VEL
LIN {X 0,Y 255.331,Z 749.21,A -85,B 0,C 180,E1 -18454.736,E2 -18454.736} C_VEL
LIN {X 0,Y 255.021,Z 746.636,A -85,B 0,C 180,E1 -18457.203,E2 -18457.203} C_VEL
LIN {X 0,Y 254.882,Z 743.233,A -85,B 0,C 180,E1 -18459.523,E2 -18459.523} C_VEL
LIN {X 0,Y 255.156,Z 738.664,A -85,B 0,C 180,E1 -18461.922,E2 -18461.922} C_VEL
LIN {X 0,Y 255.909,Z 732.913,A -85,B 0,C 180,E1 -18464.309,E2 -18464.309} C_VEL
LIN {X 0,Y 257.108,Z 725.594,A -85,B 0,C 180,E1 -18466.739,E2 -18466.739} C_VEL
LIN {X 0,Y 258.632,Z 718.588,A -85,B 0,C 180,E1 -18468.62,E2 -18468.62} C_VEL
LIN {X 0,Y 260.462,Z 709.932,A -85,B 0,C 180,E1 -18470.534,E2 -18470.534} C_VEL
LIN {X 0,Y 262.745,Z 699.303,A -85,B 0,C 180,E1 -18472.405,E2 -18472.405} C_VEL
LIN {X 0,Y 264.815,Z 688.815,A -85,B 0,C 180,E1 -18473.873,E2 -18473.873} C_VEL
LIN {X 0,Y 266.849,Z 677.341,A -85,B 0,C 180,E1 -18475.13,E2 -18475.13} C_VEL
LIN {X 0,Y 268.482,Z 665.532,A -85,B 0,C 180,E1 -18476.109,E2 -18476.109} C_VEL
LIN {X 0,Y 269.773,Z 652.458,A -85,B 0,C 180,E1 -18476.883,E2 -18476.883} C_VEL
LIN {X 0,Y 270.494,Z 639.854,A -85,B 0,C 180,E1 -18477.36,E2 -18477.36} C_VEL
LIN {X 0,Y 271.407,Z 605.97,A -85,B 0,C 180,E1 -18478.253,E2 -18478.253} C_VEL
LIN {X 0,Y 268.949,Z 577.144,A -85,B 0,C 180,E1 -18479.377,E2 -18479.377} C_VEL
LIN {X 0,Y 265.758,Z 549.333,A -85,B 0,C 180,E1 -18480.591,E2 -18480.591} C_VEL
LIN {X 0,Y 263.654,Z 533.698,A -85,B 0,C 180,E1 -18481.379,E2 -18481.379} C_VEL
LIN {X 0,Y 264.519,Z 528.928,A -85,B 0,C 180,E1 -18482.548,E2 -18482.548} C_VEL
LIN {X 0,Y 263.803,Z 523.837,A -85,B 0,C 180,E1 -18484.018,E2 -18484.018} C_VEL
LIN {X 0,Y 261.715,Z 514.111,A -85,B 0,C 180,E1 -18486.976,E2 -18486.976} C_VEL
LIN {X 0,Y 259.424,Z 504.526,A -85,B 0,C 180,E1 -18490.065,E2 -18490.065} C_VEL
LIN {X 0,Y 256.648,Z 494.484,A -85,B 0,C 180,E1 -18493.559,E2 -18493.559} C_VEL
LIN {X 0,Y 256.104,Z 492.609,A -85,B 0,C 180,E1 -18494.35,E2 -18494.35} C_VEL
LIN {X 0,Y 256.053,Z 492.582,A -85,B 0,C 180,E1 -18498.796,E2 -18498.796} C_VEL
LIN {X 0,Y 256.126,Z 492.571,A -85,B 0,C 180,E1 -18502.867,E2 -18502.867} C_VEL
LIN {X 0,Y 256.064,Z 492.568,A -85,B 0,C 180,E1 -18506.707,E2 -18506.707} C_VEL
LIN {X 0,Y 256.11,Z 492.58,A -85,B 0,C 180,E1 -18510.4,E2 -18510.4} C_VEL
LIN {X 0,Y 256.184,Z 492.558,A -85,B 0,C 180,E1 -18514.861,E2 -18514.861} C_VEL
LIN {X 0,Y 256.159,Z 492.554,A -85,B 0,C 180,E1 -18519.104,E2 -18519.104} C_VEL
LIN {X 0,Y 256.294,Z 492.552,A -85,B 0,C 180,E1 -18524.085,E2 -18524.085} C_VEL
LIN {X 0,Y 256.291,Z 492.54,A -85,B 0,C 180,E1 -18528.933,E2 -18528.933} C_VEL
LIN {X 0,Y 256.51,Z 492.533,A -85,B 0,C 180,E1 -18532.126,E2 -18532.126} C_VEL
LIN {X 0,Y 256.493,Z 492.519,A -85,B 0,C 180,E1 -18536.859,E2 -18536.859} C_VEL
LIN {X 0,Y 256.768,Z 492.5,A -85,B 0,C 180,E1 -18540,E2 -18540} C_VEL
LIN {X 0,Y 256.494,Z 492.514,A -85,B 0,C 180,E1 -18543.141,E2 -18543.141} C_VEL
LIN {X 0,Y 256.51,Z 492.522,A -85,B 0,C 180,E1 -18547.874,E2 -18547.874} C_VEL
LIN {X 0,Y 256.288,Z 492.561,A -85,B 0,C 180,E1 -18552.673,E2 -18552.673} C_VEL
LIN {X 0,Y 256.256,Z 492.545,A -85,B 0,C 180,E1 -18556.285,E2 -18556.285} C_VEL
LIN {X 0,Y 256.157,Z 492.568,A -85,B 0,C 180,E1 -18560.896,E2 -18560.896} C_VEL
LIN {X 0,Y 256.166,Z 492.577,A -85,B 0,C 180,E1 -18565.131,E2 -18565.131} C_VEL
LIN {X 0,Y 256.1,Z 492.529,A -85,B 0,C 180,E1 -18569.602,E2 -18569.602} C_VEL
LIN {X 0,Y 256.064,Z 492.56,A -85,B 0,C 180,E1 -18573.294,E2 -18573.294} C_VEL
LIN {X 0,Y 256.111,Z 492.573,A -85,B 0,C 180,E1 -18577.271,E2 -18577.271} C_VEL
LIN {X 0,Y 256.051,Z 492.551,A -85,B 0,C 180,E1 -18581.204,E2 -18581.204} C_VEL
LIN {X 0,Y 256.06,Z 492.574,A -85,B 0,C 180,E1 -18585.53,E2 -18585.53} C_VEL
LIN {X 0,Y 256.053,Z 492.568,A -85,B 0,C 180,E1 -18588.798,E2 -18588.798} C_VEL
LIN {X 0,Y 256.131,Z 492.527,A -85,B 0,C 180,E1 -18592.869,E2 -18592.869} C_VEL
LIN {X 0,Y 256.067,Z 492.511,A -85,B 0,C 180,E1 -18596.708,E2 -18596.708} C_VEL
LIN {X 0,Y 256.124,Z 492.766,A -85,B 0,C 180,E1 -18598.12,E2 -18598.12} C_VEL
LIN {X 0,Y 256.344,Z 493.732,A -85,B 0,C 180,E1 -18598.411,E2 -18598.411} C_VEL
LIN {X 0,Y 265.536,Z 510.518,A -85,B 0,C 180,E1 -18600.216,E2 -18600.216} C_VEL
LIN {X 0,Y 271.742,Z 523.399,A -85,B 0,C 180,E1 -18601.377,E2 -18601.377} C_VEL
LIN {X 0,Y 273.936,Z 528.516,A -85,B 0,C 180,E1 -18601.788,E2 -18601.788} C_VEL
LIN {X 0,Y 273.024,Z 561.681,A -85,B 0,C 180,E1 -18602.657,E2 -18602.657} C_VEL
LIN {X 0,Y 272.747,Z 580.196,A -85,B 0,C 180,E1 -18603.262,E2 -18603.262} C_VEL
LIN {X 0,Y 272.148,Z 592.758,A -85,B 0,C 180,E1 -18603.96,E2 -18603.96} C_VEL
LIN {X 0,Y 271.186,Z 604.671,A -85,B 0,C 180,E1 -18604.911,E2 -18604.911} C_VEL
LIN {X 0,Y 269.902,Z 615.929,A -85,B 0,C 180,E1 -18606.092,E2 -18606.092} C_VEL
LIN {X 0,Y 268.178,Z 626.409,A -85,B 0,C 180,E1 -18607.464,E2 -18607.464} C_VEL
LIN {X 0,Y 266.419,Z 636.501,A -85,B 0,C 180,E1 -18609.138,E2 -18609.138} C_VEL
LIN {X 0,Y 264.668,Z 645.536,A -85,B 0,C 180,E1 -18611.018,E2 -18611.018} C_VEL
LIN {X 0,Y 262.787,Z 654.293,A -85,B 0,C 180,E1 -18613.292,E2 -18613.292} C_VEL
LIN {X 0,Y 261.322,Z 660.468,A -85,B 0,C 180,E1 -18615.277,E2 -18615.277} C_VEL
LIN {X 0,Y 259.993,Z 666.074,A -85,B 0,C 180,E1 -18617.511,E2 -18617.511} C_VEL
LIN {X 0,Y 258.775,Z 670.683,A -85,B 0,C 180,E1 -18619.832,E2 -18619.832} C_VEL
LIN {X 0,Y 257.741,Z 674.219,A -85,B 0,C 180,E1 -18622.164,E2 -18622.164} C_VEL
LIN {X 0,Y 257.232,Z 676.041,A -85,B 0,C 180,E1 -18623.726,E2 -18623.726} C_VEL
LIN {X 0,Y 257.036,Z 677.382,A -85,B 0,C 180,E1 -18625.295,E2 -18625.295} C_VEL
LIN {X 0,Y 256.905,Z 678.334,A -85,B 0,C 180,E1 -18626.864,E2 -18626.864} C_VEL
LIN {X 0,Y 256.664,Z 679.162,A -85,B 0,C 180,E1 -18630,E2 -18630} C_VEL
